ABB RAPID module: P800.mod

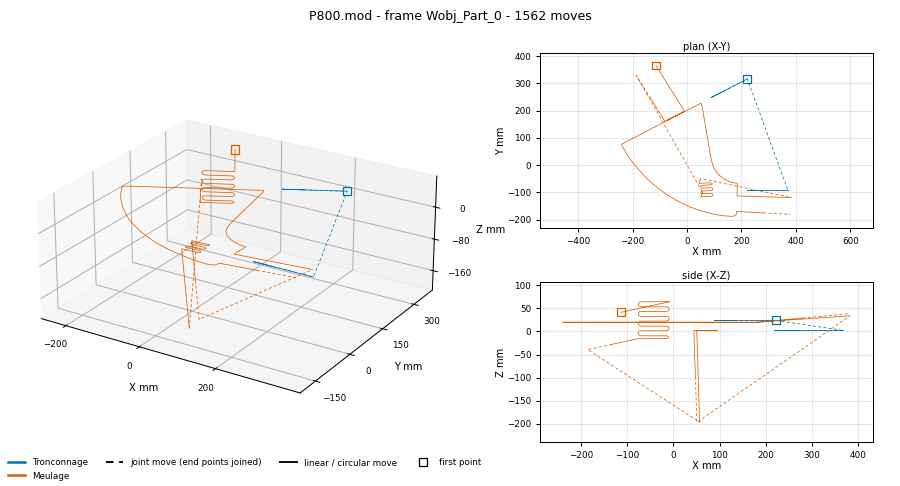
[picture p0: tool path of P800.mod in frame Wobj_Part_0, 1562 of 1576 moves have a stored position in this frame; points joined in program order, loops and branches not executed]
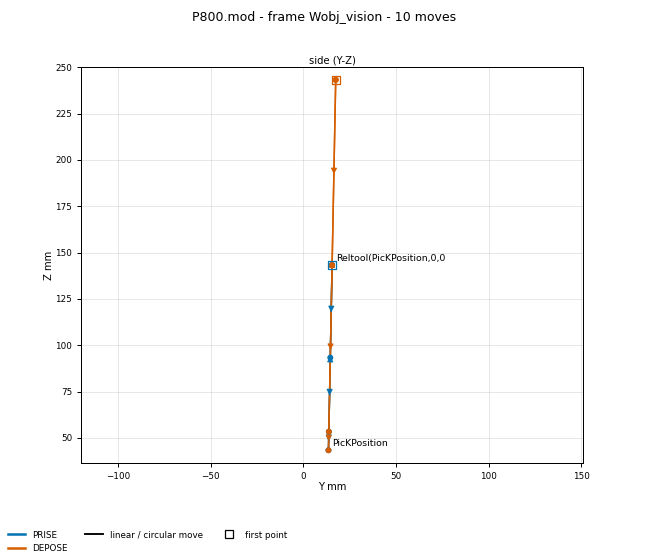
[picture p1: tool path of P800.mod in frame Wobj_vision, 10 of 1576 moves have a stored position in this frame; points joined in program order, loops and branches not executed]
MODULE P800

    ! Nom         :P800
    ! Description :
    ! Créé le     :31/05/2023 15:18:07

    LOCAL CONST SPEEDDATA VitesseLente :=[3,500,0,0];
	LOCAL CONST SPEEDDATA VitesseRapide :=[30,500,0,0];
	LOCAL CONST SPEEDDATA VitesseTronconnage :=[2,500,0,0];
	LOCAL CONST SPEEDDATA VitesseTronconnageApp :=[10,500,0,0];
    !
    !Point de prise
    LOCAL PERS Robtarget PicKPosition := [[-28.4505957143779,13.556706441967,43.2914417962046],[0.00189142649690449,0.425071382664564,-0.905103593114038,0.00991099780553871],[0,0,0,0],[8.999999E+09,8.999999E+09,8.999999E+09,8.999999E+09,8.999999E+09,8.999999E+09]];
	LOCAL PERS Pose Ref := [[0,0,0],[1,0,0,0]];
    !
    !Declaration des points de meulage

    !Tr_meulage_motif_1 : Meulage d'un motif
    LOCAL CONST Robtarget Tr_meulage_motif_1_0 := [[-8.6116181640625,197.027234375,64.58371875],[0.205457264684473,-0.183019148705642,0.639481640238406,-0.717881978735665],[0,0,0,0],[8.999999E+09,8.999999E+09,8.999999E+09,8.999999E+09,8.999999E+09,8.999999E+09]];
    LOCAL CONST Robtarget Tr_meulage_motif_1_1 := [[-9.49978125,196.567703125,64.58371875],[0.205457264684473,-0.183019148705642,0.639481640238406,-0.717881978735665],[0,0,0,0],[8.999999E+09,8.999999E+09,8.999999E+09,8.999999E+09,8.999999E+09,8.999999E+09]];
    LOCAL CONST Robtarget Tr_meulage_motif_1_2 := [[-10.3879453125,196.108171875,64.58371875],[0.205457264684473,-0.183019148705642,0.639481640238406,-0.717881978735665],[0,0,0,0],[8.999999E+09,8.999999E+09,8.999999E+09,8.999999E+09,8.999999E+09,8.999999E+09]];
    LOCAL CONST Robtarget Tr_meulage_motif_1_3 := [[-11.276109375,195.648640625,64.58371875],[0.205457264684473,-0.183019148705642,0.639481640238406,-0.717881978735665],[0,0,0,0],[8.999999E+09,8.999999E+09,8.999999E+09,8.999999E+09,8.999999E+09,8.999999E+09]];
    LOCAL CONST Robtarget Tr_meulage_motif_1_4 := [[-12.1642724609375,195.189125,64.58372265625],[0.205457264684473,-0.183019148705642,0.639481640238406,-0.717881978735665],[0,0,0,0],[8.999999E+09,8.999999E+09,8.999999E+09,8.999999E+09,8.999999E+09,8.999999E+09]];
    LOCAL CONST Robtarget Tr_meulage_motif_1_5 := [[-13.0524365234375,194.72959375,64.58372265625],[0.205457264684473,-0.183019148705642,0.639481640238406,-0.717881978735665],[0,0,0,0],[8.999999E+09,8.999999E+09,8.999999E+09,8.999999E+09,8.999999E+09,8.999999E+09]];
    LOCAL CONST Robtarget Tr_meulage_motif_1_6 := [[-13.940599609375,194.2700625,64.58372265625],[0.205457264684473,-0.183019148705642,0.639481640238406,-0.717881978735665],[0,0,0,0],[8.999999E+09,8.999999E+09,8.999999E+09,8.999999E+09,8.999999E+09,8.999999E+09]];
    LOCAL CONST Robtarget Tr_meulage_motif_1_7 := [[-14.828763671875,193.81053125,64.58372265625],[0.205457264684473,-0.183019148705642,0.639481640238406,-0.717881978735665],[0,0,0,0],[8.999999E+09,8.999999E+09,8.999999E+09,8.999999E+09,8.999999E+09,8.999999E+09]];
    LOCAL CONST Robtarget Tr_meulage_motif_1_8 := [[-15.7169267578125,193.351015625,64.58372265625],[0.205457264684473,-0.183019148705642,0.639481640238406,-0.717881978735665],[0,0,0,0],[8.999999E+09,8.999999E+09,8.999999E+09,8.999999E+09,8.999999E+09,8.999999E+09]];
    LOCAL CONST Robtarget Tr_meulage_motif_1_9 := [[-16.60508984375,192.891484375,64.58372265625],[0.205457264684473,-0.183019148705642,0.639481640238406,-0.717881978735665],[0,0,0,0],[8.999999E+09,8.999999E+09,8.999999E+09,8.999999E+09,8.999999E+09,8.999999E+09]];
    LOCAL CONST Robtarget Tr_meulage_motif_1_10 := [[-17.49325390625,192.431953125,64.58372265625],[0.205457264684473,-0.183019148705642,0.639481640238406,-0.717881978735665],[0,0,0,0],[8.999999E+09,8.999999E+09,8.999999E+09,8.999999E+09,8.999999E+09,8.999999E+09]];
    LOCAL CONST Robtarget Tr_meulage_motif_1_11 := [[-18.38141796875,191.972421875,64.58372265625],[0.205457264684473,-0.183019148705642,0.639481640238406,-0.717881978735665],[0,0,0,0],[8.999999E+09,8.999999E+09,8.999999E+09,8.999999E+09,8.999999E+09,8.999999E+09]];
    LOCAL CONST Robtarget Tr_meulage_motif_1_12 := [[-19.26958203125,191.51290625,64.5837265625],[0.205457264684473,-0.183019148705642,0.639481640238406,-0.717881978735665],[0,0,0,0],[8.999999E+09,8.999999E+09,8.999999E+09,8.999999E+09,8.999999E+09,8.999999E+09]];
    LOCAL CONST Robtarget Tr_meulage_motif_1_13 := [[-20.157744140625,191.053375,64.5837265625],[0.205457264684473,-0.183019148705642,0.639481640238406,-0.717881978735665],[0,0,0,0],[8.999999E+09,8.999999E+09,8.999999E+09,8.999999E+09,8.999999E+09,8.999999E+09]];
    LOCAL CONST Robtarget Tr_meulage_motif_1_14 := [[-21.045908203125,190.59384375,64.5837265625],[0.205457264684473,-0.183019148705642,0.639481640238406,-0.717881978735665],[0,0,0,0],[8.999999E+09,8.999999E+09,8.999999E+09,8.999999E+09,8.999999E+09,8.999999E+09]];
    LOCAL CONST Robtarget Tr_meulage_motif_1_15 := [[-21.934072265625,190.1343125,64.5837265625],[0.205457264684473,-0.183019148705642,0.639481640238406,-0.717881978735665],[0,0,0,0],[8.999999E+09,8.999999E+09,8.999999E+09,8.999999E+09,8.999999E+09,8.999999E+09]];
    LOCAL CONST Robtarget Tr_meulage_motif_1_16 := [[-22.822236328125,189.674796875,64.5837265625],[0.205457264684473,-0.183019148705642,0.639481640238406,-0.717881978735665],[0,0,0,0],[8.999999E+09,8.999999E+09,8.999999E+09,8.999999E+09,8.999999E+09,8.999999E+09]];
    LOCAL CONST Robtarget Tr_meulage_motif_1_17 := [[-23.7103984375,189.215265625,64.5837265625],[0.205457264684473,-0.183019148705642,0.639481640238406,-0.717881978735665],[0,0,0,0],[8.999999E+09,8.999999E+09,8.999999E+09,8.999999E+09,8.999999E+09,8.999999E+09]];
    LOCAL CONST Robtarget Tr_meulage_motif_1_18 := [[-24.5985625,188.755734375,64.5837265625],[0.205457264684473,-0.183019148705642,0.639481640238406,-0.717881978735665],[0,0,0,0],[8.999999E+09,8.999999E+09,8.999999E+09,8.999999E+09,8.999999E+09,8.999999E+09]];
    LOCAL CONST Robtarget Tr_meulage_motif_1_19 := [[-25.4867265625,188.296203125,64.5837265625],[0.205457264684473,-0.183019148705642,0.639481640238406,-0.717881978735665],[0,0,0,0],[8.999999E+09,8.999999E+09,8.999999E+09,8.999999E+09,8.999999E+09,8.999999E+09]];
    LOCAL CONST Robtarget Tr_meulage_motif_1_20 := [[-26.374890625,187.8366875,64.5837265625],[0.205457264684473,-0.183019148705642,0.639481640238406,-0.717881978735665],[0,0,0,0],[8.999999E+09,8.999999E+09,8.999999E+09,8.999999E+09,8.999999E+09,8.999999E+09]];
    LOCAL CONST Robtarget Tr_meulage_motif_1_21 := [[-27.263052734375,187.37715625,64.58373046875],[0.205457264684473,-0.183019148705642,0.639481640238406,-0.717881978735665],[0,0,0,0],[8.999999E+09,8.999999E+09,8.999999E+09,8.999999E+09,8.999999E+09,8.999999E+09]];
    LOCAL CONST Robtarget Tr_meulage_motif_1_22 := [[-28.151216796875,186.917625,64.58373046875],[0.205457264684473,-0.183019148705642,0.639481640238406,-0.717881978735665],[0,0,0,0],[8.999999E+09,8.999999E+09,8.999999E+09,8.999999E+09,8.999999E+09,8.999999E+09]];
    LOCAL CONST Robtarget Tr_meulage_motif_1_23 := [[-29.039380859375,186.45809375,64.58373046875],[0.205457264684473,-0.183019148705642,0.639481640238406,-0.717881978735665],[0,0,0,0],[8.999999E+09,8.999999E+09,8.999999E+09,8.999999E+09,8.999999E+09,8.999999E+09]];
    LOCAL CONST Robtarget Tr_meulage_motif_1_24 := [[-29.927544921875,185.9985625,64.58373046875],[0.205457264684473,-0.183019148705642,0.639481640238406,-0.717881978735665],[0,0,0,0],[8.999999E+09,8.999999E+09,8.999999E+09,8.999999E+09,8.999999E+09,8.999999E+09]];
    LOCAL CONST Robtarget Tr_meulage_motif_1_25 := [[-30.815708984375,185.539046875,64.58373046875],[0.205457264684473,-0.183019148705642,0.639481640238406,-0.717881978735665],[0,0,0,0],[8.999999E+09,8.999999E+09,8.999999E+09,8.999999E+09,8.999999E+09,8.999999E+09]];
    LOCAL CONST Robtarget Tr_meulage_motif_1_26 := [[-31.70387109375,185.079515625,64.58373046875],[0.205457264684473,-0.183019148705642,0.639481640238406,-0.717881978735665],[0,0,0,0],[8.999999E+09,8.999999E+09,8.999999E+09,8.999999E+09,8.999999E+09,8.999999E+09]];
    LOCAL CONST Robtarget Tr_meulage_motif_1_27 := [[-32.59203515625,184.619984375,64.58373046875],[0.205457264684473,-0.183019148705642,0.639481640238406,-0.717881978735665],[0,0,0,0],[8.999999E+09,8.999999E+09,8.999999E+09,8.999999E+09,8.999999E+09,8.999999E+09]];
    LOCAL CONST Robtarget Tr_meulage_motif_1_28 := [[-33.48019921875,184.160453125,64.58373046875],[0.205457264684473,-0.183019148705642,0.639481640238406,-0.717881978735665],[0,0,0,0],[8.999999E+09,8.999999E+09,8.999999E+09,8.999999E+09,8.999999E+09,8.999999E+09]];
    LOCAL CONST Robtarget Tr_meulage_motif_1_29 := [[-34.36836328125,183.7009375,64.583734375],[0.205457264684473,-0.183019148705642,0.639481640238406,-0.717881978735665],[0,0,0,0],[8.999999E+09,8.999999E+09,8.999999E+09,8.999999E+09,8.999999E+09,8.999999E+09]];
    LOCAL CONST Robtarget Tr_meulage_motif_1_30 := [[-35.25652734375,183.24140625,64.583734375],[0.205457264684473,-0.183019148705642,0.639481640238406,-0.717881978735665],[0,0,0,0],[8.999999E+09,8.999999E+09,8.999999E+09,8.999999E+09,8.999999E+09,8.999999E+09]];
    LOCAL CONST Robtarget Tr_meulage_motif_1_31 := [[-36.14469140625,182.781875,64.583734375],[0.205457264684473,-0.183019148705642,0.639481640238406,-0.717881978735665],[0,0,0,0],[8.999999E+09,8.999999E+09,8.999999E+09,8.999999E+09,8.999999E+09,8.999999E+09]];
    LOCAL CONST Robtarget Tr_meulage_motif_1_32 := [[-37.0328515625,182.32234375,64.583734375],[0.205457264684473,-0.183019148705642,0.639481640238406,-0.717881978735665],[0,0,0,0],[8.999999E+09,8.999999E+09,8.999999E+09,8.999999E+09,8.999999E+09,8.999999E+09]];
    LOCAL CONST Robtarget Tr_meulage_motif_1_33 := [[-37.921015625,181.862828125,64.583734375],[0.205457264684473,-0.183019148705642,0.639481640238406,-0.717881978735665],[0,0,0,0],[8.999999E+09,8.999999E+09,8.999999E+09,8.999999E+09,8.999999E+09,8.999999E+09]];
    LOCAL CONST Robtarget Tr_meulage_motif_1_34 := [[-38.8091796875,181.403296875,64.583734375],[0.205457264684473,-0.183019148705642,0.639481640238406,-0.717881978735665],[0,0,0,0],[8.999999E+09,8.999999E+09,8.999999E+09,8.999999E+09,8.999999E+09,8.999999E+09]];
    LOCAL CONST Robtarget Tr_meulage_motif_1_35 := [[-39.69734375,180.943765625,64.583734375],[0.205457264684473,-0.183019148705642,0.639481640238406,-0.717881978735665],[0,0,0,0],[8.999999E+09,8.999999E+09,8.999999E+09,8.999999E+09,8.999999E+09,8.999999E+09]];
    LOCAL CONST Robtarget Tr_meulage_motif_1_36 := [[-40.5855078125,180.484234375,64.583734375],[0.205457264684473,-0.183019148705642,0.639481640238406,-0.717881978735665],[0,0,0,0],[8.999999E+09,8.999999E+09,8.999999E+09,8.999999E+09,8.999999E+09,8.999999E+09]];
    LOCAL CONST Robtarget Tr_meulage_motif_1_37 := [[-41.473671875,180.02471875,64.583734375],[0.205457264684473,-0.183019148705642,0.639481640238406,-0.717881978735665],[0,0,0,0],[8.999999E+09,8.999999E+09,8.999999E+09,8.999999E+09,8.999999E+09,8.999999E+09]];
    LOCAL CONST Robtarget Tr_meulage_motif_1_38 := [[-42.3618359375,179.5651875,64.58373828125],[0.205457264684473,-0.183019148705642,0.639481640238406,-0.717881978735665],[0,0,0,0],[8.999999E+09,8.999999E+09,8.999999E+09,8.999999E+09,8.999999E+09,8.999999E+09]];
    LOCAL CONST Robtarget Tr_meulage_motif_1_39 := [[-43.25,179.10565625,64.58373828125],[0.205457264684473,-0.183019148705642,0.639481640238406,-0.717881978735665],[0,0,0,0],[8.999999E+09,8.999999E+09,8.999999E+09,8.999999E+09,8.999999E+09,8.999999E+09]];
    LOCAL CONST Robtarget Tr_meulage_motif_1_40 := [[-44.13816015625,178.646125,64.58373828125],[0.205457264684473,-0.183019148705642,0.639481640238406,-0.717881978735665],[0,0,0,0],[8.999999E+09,8.999999E+09,8.999999E+09,8.999999E+09,8.999999E+09,8.999999E+09]];
    LOCAL CONST Robtarget Tr_meulage_motif_1_41 := [[-45.02632421875,178.186609375,64.58373828125],[0.205457264684473,-0.183019148705642,0.639481640238406,-0.717881978735665],[0,0,0,0],[8.999999E+09,8.999999E+09,8.999999E+09,8.999999E+09,8.999999E+09,8.999999E+09]];
    LOCAL CONST Robtarget Tr_meulage_motif_1_42 := [[-45.91448828125,177.727078125,64.58373828125],[0.205457264684473,-0.183019148705642,0.639481640238406,-0.717881978735665],[0,0,0,0],[8.999999E+09,8.999999E+09,8.999999E+09,8.999999E+09,8.999999E+09,8.999999E+09]];
    LOCAL CONST Robtarget Tr_meulage_motif_1_43 := [[-46.80265234375,177.267546875,64.58373828125],[0.205457264684473,-0.183019148705642,0.639481640238406,-0.717881978735665],[0,0,0,0],[8.999999E+09,8.999999E+09,8.999999E+09,8.999999E+09,8.999999E+09,8.999999E+09]];
    LOCAL CONST Robtarget Tr_meulage_motif_1_44 := [[-47.69081640625,176.808015625,64.58373828125],[0.205457264684473,-0.183019148705642,0.639481640238406,-0.717881978735665],[0,0,0,0],[8.999999E+09,8.999999E+09,8.999999E+09,8.999999E+09,8.999999E+09,8.999999E+09]];
    LOCAL CONST Robtarget Tr_meulage_motif_1_45 := [[-48.57898046875,176.3485,64.58373828125],[0.205457264684473,-0.183019148705642,0.639481640238406,-0.717881978735665],[0,0,0,0],[8.999999E+09,8.999999E+09,8.999999E+09,8.999999E+09,8.999999E+09,8.999999E+09]];
    LOCAL CONST Robtarget Tr_meulage_motif_1_46 := [[-49.46714453125,175.88896875,64.5837421875],[0.205457264684473,-0.183019148705642,0.639481640238406,-0.717881978735665],[0,0,0,0],[8.999999E+09,8.999999E+09,8.999999E+09,8.999999E+09,8.999999E+09,8.999999E+09]];
    LOCAL CONST Robtarget Tr_meulage_motif_1_47 := [[-50.35530859375,175.4294375,64.5837421875],[0.205457264684473,-0.183019148705642,0.639481640238406,-0.717881978735665],[0,0,0,0],[8.999999E+09,8.999999E+09,8.999999E+09,8.999999E+09,8.999999E+09,8.999999E+09]];
    LOCAL CONST Robtarget Tr_meulage_motif_1_48 := [[-51.24347265625,174.96990625,64.5837421875],[0.205457264684473,-0.183019148705642,0.639481640238406,-0.717881978735665],[0,0,0,0],[8.999999E+09,8.999999E+09,8.999999E+09,8.999999E+09,8.999999E+09,8.999999E+09]];
    LOCAL CONST Robtarget Tr_meulage_motif_1_49 := [[-52.1316328125,174.510390625,64.5837421875],[0.205457264684473,-0.183019148705642,0.639481640238406,-0.717881978735665],[0,0,0,0],[8.999999E+09,8.999999E+09,8.999999E+09,8.999999E+09,8.999999E+09,8.999999E+09]];
    LOCAL CONST Robtarget Tr_meulage_motif_1_50 := [[-53.019796875,174.050859375,64.5837421875],[0.205457264684473,-0.183019148705642,0.639481640238406,-0.717881978735665],[0,0,0,0],[8.999999E+09,8.999999E+09,8.999999E+09,8.999999E+09,8.999999E+09,8.999999E+09]];
    LOCAL CONST Robtarget Tr_meulage_motif_1_51 := [[-53.9079609375,173.591328125,64.5837421875],[0.205457264684473,-0.183019148705642,0.639481640238406,-0.717881978735665],[0,0,0,0],[8.999999E+09,8.999999E+09,8.999999E+09,8.999999E+09,8.999999E+09,8.999999E+09]];
    LOCAL CONST Robtarget Tr_meulage_motif_1_52 := [[-54.796125,173.131796875,64.5837421875],[0.205457264684473,-0.183019148705642,0.639481640238406,-0.717881978735665],[0,0,0,0],[8.999999E+09,8.999999E+09,8.999999E+09,8.999999E+09,8.999999E+09,8.999999E+09]];
    LOCAL CONST Robtarget Tr_meulage_motif_1_53 := [[-55.6842890625,172.67228125,64.5837421875],[0.205457264684473,-0.183019148705642,0.639481640238406,-0.717881978735665],[0,0,0,0],[8.999999E+09,8.999999E+09,8.999999E+09,8.999999E+09,8.999999E+09,8.999999E+09]];
    LOCAL CONST Robtarget Tr_meulage_motif_1_54 := [[-56.572453125,172.21275,64.5837421875],[0.205457264684473,-0.183019148705642,0.639481640238406,-0.717881978735665],[0,0,0,0],[8.999999E+09,8.999999E+09,8.999999E+09,8.999999E+09,8.999999E+09,8.999999E+09]];
    LOCAL CONST Robtarget Tr_meulage_motif_1_55 := [[-57.4606171875,171.75321875,64.58374609375],[0.205457264684473,-0.183019148705642,0.639481640238406,-0.717881978735665],[0,0,0,0],[8.999999E+09,8.999999E+09,8.999999E+09,8.999999E+09,8.999999E+09,8.999999E+09]];
    LOCAL CONST Robtarget Tr_meulage_motif_1_56 := [[-58.34878125,171.2936875,64.58374609375],[0.205457264684473,-0.183019148705642,0.639481640238406,-0.717881978735665],[0,0,0,0],[8.999999E+09,8.999999E+09,8.999999E+09,8.999999E+09,8.999999E+09,8.999999E+09]];
    LOCAL CONST Robtarget Tr_meulage_motif_1_57 := [[-59.23694140625,170.834171875,64.58374609375],[0.205457264684473,-0.183019148705642,0.639481640238406,-0.717881978735665],[0,0,0,0],[8.999999E+09,8.999999E+09,8.999999E+09,8.999999E+09,8.999999E+09,8.999999E+09]];
    LOCAL CONST Robtarget Tr_meulage_motif_1_58 := [[-60.12510546875,170.374640625,64.58374609375],[0.205457264684473,-0.183019148705642,0.639481640238406,-0.717881978735665],[0,0,0,0],[8.999999E+09,8.999999E+09,8.999999E+09,8.999999E+09,8.999999E+09,8.999999E+09]];
    LOCAL CONST Robtarget Tr_meulage_motif_1_59 := [[-61.01326953125,169.915109375,64.58374609375],[0.205457264684473,-0.183019148705642,0.639481640238406,-0.717881978735665],[0,0,0,0],[8.999999E+09,8.999999E+09,8.999999E+09,8.999999E+09,8.999999E+09,8.999999E+09]];
    LOCAL CONST Robtarget Tr_meulage_motif_1_60 := [[-61.90143359375,169.455578125,64.58374609375],[0.205457264684473,-0.183019148705642,0.639481640238406,-0.717881978735665],[0,0,0,0],[8.999999E+09,8.999999E+09,8.999999E+09,8.999999E+09,8.999999E+09,8.999999E+09]];
    LOCAL CONST Robtarget Tr_meulage_motif_1_61 := [[-62.78959765625,168.9960625,64.58374609375],[0.205457264684473,-0.183019148705642,0.639481640238406,-0.717881978735665],[0,0,0,0],[8.999999E+09,8.999999E+09,8.999999E+09,8.999999E+09,8.999999E+09,8.999999E+09]];
    LOCAL CONST Robtarget Tr_meulage_motif_1_62 := [[-63.67776171875,168.53653125,64.58374609375],[0.205457264684473,-0.183019148705642,0.639481640238406,-0.717881978735665],[0,0,0,0],[8.999999E+09,8.999999E+09,8.999999E+09,8.999999E+09,8.999999E+09,8.999999E+09]];
    LOCAL CONST Robtarget Tr_meulage_motif_1_63 := [[-64.56592578125,168.077,64.58374609375],[0.205457264684473,-0.183019148705642,0.639481640238406,-0.717881978735665],[0,0,0,0],[8.999999E+09,8.999999E+09,8.999999E+09,8.999999E+09,8.999999E+09,8.999999E+09]];
    LOCAL CONST Robtarget Tr_meulage_motif_1_64 := [[-65.45408984375,167.61746875,64.58375],[0.205457264684473,-0.183019148705642,0.639481640238406,-0.717881978735665],[0,0,0,0],[8.999999E+09,8.999999E+09,8.999999E+09,8.999999E+09,8.999999E+09,8.999999E+09]];
    LOCAL CONST Robtarget Tr_meulage_motif_1_65 := [[-66.34225,167.157953125,64.58375],[0.205457264684473,-0.183019148705642,0.639481640238406,-0.717881978735665],[0,0,0,0],[8.999999E+09,8.999999E+09,8.999999E+09,8.999999E+09,8.999999E+09,8.999999E+09]];
    LOCAL CONST Robtarget Tr_meulage_motif_1_66 := [[-67.2304140625,166.698421875,64.58375],[0.205457264684473,-0.183019148705642,0.639481640238406,-0.717881978735665],[0,0,0,0],[8.999999E+09,8.999999E+09,8.999999E+09,8.999999E+09,8.999999E+09,8.999999E+09]];
    LOCAL CONST Robtarget Tr_meulage_motif_1_67 := [[-68.118578125,166.238890625,64.58375],[0.205457264684473,-0.183019148705642,0.639481640238406,-0.717881978735665],[0,0,0,0],[8.999999E+09,8.999999E+09,8.999999E+09,8.999999E+09,8.999999E+09,8.999999E+09]];
    LOCAL CONST Robtarget Tr_meulage_motif_1_68 := [[-69.0067421875,165.779359375,64.58375],[0.205457264684473,-0.183019148705642,0.639481640238406,-0.717881978735665],[0,0,0,0],[8.999999E+09,8.999999E+09,8.999999E+09,8.999999E+09,8.999999E+09,8.999999E+09]];
    LOCAL CONST Robtarget Tr_meulage_motif_1_69 := [[-69.89490625,165.31984375,64.58375],[0.205457264684473,-0.183019148705642,0.639481640238406,-0.717881978735665],[0,0,0,0],[8.999999E+09,8.999999E+09,8.999999E+09,8.999999E+09,8.999999E+09,8.999999E+09]];
    LOCAL CONST Robtarget Tr_meulage_motif_1_70 := [[-70.7768671875,164.864515625,64.47316015625],[0.205457264684473,-0.183019148705642,0.639481640238406,-0.717881978735665],[0,0,0,0],[8.999999E+09,8.999999E+09,8.999999E+09,8.999999E+09,8.999999E+09,8.999999E+09]];
    LOCAL CONST Robtarget Tr_meulage_motif_1_71 := [[-71.6182890625,164.4310625,64.26198046875],[0.205457264684473,-0.183019148705642,0.639481640238406,-0.717881978735665],[0,0,0,0],[8.999999E+09,8.999999E+09,8.999999E+09,8.999999E+09,8.999999E+09,8.999999E+09]];
    LOCAL CONST Robtarget Tr_meulage_motif_1_72 := [[-72.376640625,164.041140625,63.99014453125],[0.205457264684473,-0.183019148705642,0.639481640238406,-0.717881978735665],[0,0,0,0],[8.999999E+09,8.999999E+09,8.999999E+09,8.999999E+09,8.999999E+09,8.999999E+09]];
    LOCAL CONST Robtarget Tr_meulage_motif_1_73 := [[-73.0436875,163.698484375,63.71421875],[0.205457264684473,-0.183019148705642,0.639481640238406,-0.717881978735665],[0,0,0,0],[8.999999E+09,8.999999E+09,8.999999E+09,8.999999E+09,8.999999E+09,8.999999E+09]];
    LOCAL CONST Robtarget Tr_meulage_motif_1_74 := [[-74.0238984375,163.196859375,63.09811328125],[0.205457264684473,-0.183019148705642,0.639481640238406,-0.717881978735665],[0,0,0,0],[8.999999E+09,8.999999E+09,8.999999E+09,8.999999E+09,8.999999E+09,8.999999E+09]];
    LOCAL CONST Robtarget Tr_meulage_motif_1_75 := [[-74.9363671875,162.732359375,62.250484375],[0.205457264684473,-0.183019148705642,0.639481640238406,-0.717881978735665],[0,0,0,0],[8.999999E+09,8.999999E+09,8.999999E+09,8.999999E+09,8.999999E+09,8.999999E+09]];
    LOCAL CONST Robtarget Tr_meulage_motif_1_76 := [[-75.6929765625,162.35009375,61.226640625],[0.205457264684473,-0.183019148705642,0.639481640238406,-0.717881978735665],[0,0,0,0],[8.999999E+09,8.999999E+09,8.999999E+09,8.999999E+09,8.999999E+09,8.999999E+09]];
    LOCAL CONST Robtarget Tr_meulage_motif_1_77 := [[-76.130625,162.133671875,60.11048828125],[0.205457264684473,-0.183019148705642,0.639481640238406,-0.717881978735665],[0,0,0,0],[8.999999E+09,8.999999E+09,8.999999E+09,8.999999E+09,8.999999E+09,8.999999E+09]];
    LOCAL CONST Robtarget Tr_meulage_motif_1_78 := [[-76.1572109375,162.12615625,59.41454296875],[0.205457264684473,-0.183019148705642,0.639481640238406,-0.717881978735665],[0,0,0,0],[8.999999E+09,8.999999E+09,8.999999E+09,8.999999E+09,8.999999E+09,8.999999E+09]];
    LOCAL CONST Robtarget Tr_meulage_motif_1_79 := [[-76.1596328125,162.130828125,58.7533125],[0.205457264684473,-0.183019148705642,0.639481640238406,-0.717881978735665],[0,0,0,0],[8.999999E+09,8.999999E+09,8.999999E+09,8.999999E+09,8.999999E+09,8.999999E+09]];
    LOCAL CONST Robtarget Tr_meulage_motif_1_80 := [[-76.1133125,162.160734375,58.0922421875],[0.205457264684473,-0.183019148705642,0.639481640238406,-0.717881978735665],[0,0,0,0],[8.999999E+09,8.999999E+09,8.999999E+09,8.999999E+09,8.999999E+09,8.999999E+09]];
    LOCAL CONST Robtarget Tr_meulage_motif_1_81 := [[-75.67484375,162.39746875,56.99052734375],[0.205457264684473,-0.183019148705642,0.639481640238406,-0.717881978735665],[0,0,0,0],[8.999999E+09,8.999999E+09,8.999999E+09,8.999999E+09,8.999999E+09,8.999999E+09]];
    LOCAL CONST Robtarget Tr_meulage_motif_1_82 := [[-74.9177109375,162.798234375,55.98393359375],[0.205457264684473,-0.183019148705642,0.639481640238406,-0.717881978735665],[0,0,0,0],[8.999999E+09,8.999999E+09,8.999999E+09,8.999999E+09,8.999999E+09,8.999999E+09]];
    LOCAL CONST Robtarget Tr_meulage_motif_1_83 := [[-74.011765625,163.274390625,55.15508203125],[0.205457264684473,-0.183019148705642,0.639481640238406,-0.717881978735665],[0,0,0,0],[8.999999E+09,8.999999E+09,8.999999E+09,8.999999E+09,8.999999E+09,8.999999E+09]];
    LOCAL CONST Robtarget Tr_meulage_motif_1_84 := [[-73.4029921875,163.592921875,54.75934375],[0.205457264684473,-0.183019148705642,0.639481640238406,-0.717881978735665],[0,0,0,0],[8.999999E+09,8.999999E+09,8.999999E+09,8.999999E+09,8.999999E+09,8.999999E+09]];
    LOCAL CONST Robtarget Tr_meulage_motif_1_85 := [[-72.376140625,164.128578125,54.271828125],[0.205457264684473,-0.183019148705642,0.639481640238406,-0.717881978735665],[0,0,0,0],[8.999999E+09,8.999999E+09,8.999999E+09,8.999999E+09,8.999999E+09,8.999999E+09]];
    LOCAL CONST Robtarget Tr_meulage_motif_1_86 := [[-71.6265859375,164.518765625,54.0077421875],[0.205457264684473,-0.183019148705642,0.639481640238406,-0.717881978735665],[0,0,0,0],[8.999999E+09,8.999999E+09,8.999999E+09,8.999999E+09,8.999999E+09,8.999999E+09]];
    LOCAL CONST Robtarget Tr_meulage_motif_1_87 := [[-70.7995625,164.948484375,53.80328125],[0.205457264684473,-0.183019148705642,0.639481640238406,-0.717881978735665],[0,0,0,0],[8.999999E+09,8.999999E+09,8.999999E+09,8.999999E+09,8.999999E+09,8.999999E+09]];
    LOCAL CONST Robtarget Tr_meulage_motif_1_88 := [[-69.928171875,165.4003125,53.69469140625],[0.205457264684473,-0.183019148705642,0.639481640238406,-0.717881978735665],[0,0,0,0],[8.999999E+09,8.999999E+09,8.999999E+09,8.999999E+09,8.999999E+09,8.999999E+09]];
    LOCAL CONST Robtarget Tr_meulage_motif_1_89 := [[-69.0470234375,165.857203125,53.58409765625],[0.205457264684473,-0.183019148705642,0.639481640238406,-0.717881978735665],[0,0,0,0],[8.999999E+09,8.999999E+09,8.999999E+09,8.999999E+09,8.999999E+09,8.999999E+09]];
    LOCAL CONST Robtarget Tr_meulage_motif_1_90 := [[-68.158859375,166.316734375,53.58409765625],[0.205457264684473,-0.183019148705642,0.639481640238406,-0.717881978735665],[0,0,0,0],[8.999999E+09,8.999999E+09,8.999999E+09,8.999999E+09,8.999999E+09,8.999999E+09]];
    LOCAL CONST Robtarget Tr_meulage_motif_1_91 := [[-67.2706953125,166.77625,53.58409765625],[0.205457264684473,-0.183019148705642,0.639481640238406,-0.717881978735665],[0,0,0,0],[8.999999E+09,8.999999E+09,8.999999E+09,8.999999E+09,8.999999E+09,8.999999E+09]];
    LOCAL CONST Robtarget Tr_meulage_motif_1_92 := [[-66.38253125,167.23578125,53.58409765625],[0.205457264684473,-0.183019148705642,0.639481640238406,-0.717881978735665],[0,0,0,0],[8.999999E+09,8.999999E+09,8.999999E+09,8.999999E+09,8.999999E+09,8.999999E+09]];
    LOCAL CONST Robtarget Tr_meulage_motif_1_93 := [[-65.4943671875,167.6953125,53.58409765625],[0.205457264684473,-0.183019148705642,0.639481640238406,-0.717881978735665],[0,0,0,0],[8.999999E+09,8.999999E+09,8.999999E+09,8.999999E+09,8.999999E+09,8.999999E+09]];
    LOCAL CONST Robtarget Tr_meulage_motif_1_94 := [[-64.606203125,168.15484375,53.58409765625],[0.205457264684473,-0.183019148705642,0.639481640238406,-0.717881978735665],[0,0,0,0],[8.999999E+09,8.999999E+09,8.999999E+09,8.999999E+09,8.999999E+09,8.999999E+09]];
    LOCAL CONST Robtarget Tr_meulage_motif_1_95 := [[-63.7180390625,168.614359375,53.58409765625],[0.205457264684473,-0.183019148705642,0.639481640238406,-0.717881978735665],[0,0,0,0],[8.999999E+09,8.999999E+09,8.999999E+09,8.999999E+09,8.999999E+09,8.999999E+09]];
    LOCAL CONST Robtarget Tr_meulage_motif_1_96 := [[-62.829875,169.073890625,53.58409765625],[0.205457264684473,-0.183019148705642,0.639481640238406,-0.717881978735665],[0,0,0,0],[8.999999E+09,8.999999E+09,8.999999E+09,8.999999E+09,8.999999E+09,8.999999E+09]];
    LOCAL CONST Robtarget Tr_meulage_motif_1_97 := [[-61.9417109375,169.533421875,53.58409765625],[0.205457264684473,-0.183019148705642,0.639481640238406,-0.717881978735665],[0,0,0,0],[8.999999E+09,8.999999E+09,8.999999E+09,8.999999E+09,8.999999E+09,8.999999E+09]];
    LOCAL CONST Robtarget Tr_meulage_motif_1_98 := [[-61.053546875,169.992953125,53.58409375],[0.205457264684473,-0.183019148705642,0.639481640238406,-0.717881978735665],[0,0,0,0],[8.999999E+09,8.999999E+09,8.999999E+09,8.999999E+09,8.999999E+09,8.999999E+09]];
    LOCAL CONST Robtarget Tr_meulage_motif_1_99 := [[-60.1653828125,170.45246875,53.58409375],[0.205457264684473,-0.183019148705642,0.639481640238406,-0.717881978735665],[0,0,0,0],[8.999999E+09,8.999999E+09,8.999999E+09,8.999999E+09,8.999999E+09,8.999999E+09]];
    LOCAL CONST Robtarget Tr_meulage_motif_1_100 := [[-59.27721875,170.912,53.58409375],[0.205457264684473,-0.183019148705642,0.639481640238406,-0.717881978735665],[0,0,0,0],[8.999999E+09,8.999999E+09,8.999999E+09,8.999999E+09,8.999999E+09,8.999999E+09]];
    LOCAL CONST Robtarget Tr_meulage_motif_1_101 := [[-58.38905859375,171.37153125,53.58409375],[0.205457264684473,-0.183019148705642,0.639481640238406,-0.717881978735665],[0,0,0,0],[8.999999E+09,8.999999E+09,8.999999E+09,8.999999E+09,8.999999E+09,8.999999E+09]];
    LOCAL CONST Robtarget Tr_meulage_motif_1_102 := [[-57.50089453125,171.8310625,53.58409375],[0.205457264684473,-0.183019148705642,0.639481640238406,-0.717881978735665],[0,0,0,0],[8.999999E+09,8.999999E+09,8.999999E+09,8.999999E+09,8.999999E+09,8.999999E+09]];
    LOCAL CONST Robtarget Tr_meulage_motif_1_103 := [[-56.61273046875,172.290578125,53.58409375],[0.205457264684473,-0.183019148705642,0.639481640238406,-0.717881978735665],[0,0,0,0],[8.999999E+09,8.999999E+09,8.999999E+09,8.999999E+09,8.999999E+09,8.999999E+09]];
    LOCAL CONST Robtarget Tr_meulage_motif_1_104 := [[-55.72456640625,172.750109375,53.58409375],[0.205457264684473,-0.183019148705642,0.639481640238406,-0.717881978735665],[0,0,0,0],[8.999999E+09,8.999999E+09,8.999999E+09,8.999999E+09,8.999999E+09,8.999999E+09]];
    LOCAL CONST Robtarget Tr_meulage_motif_1_105 := [[-54.83640234375,173.209640625,53.58409375],[0.205457264684473,-0.183019148705642,0.639481640238406,-0.717881978735665],[0,0,0,0],[8.999999E+09,8.999999E+09,8.999999E+09,8.999999E+09,8.999999E+09,8.999999E+09]];
    LOCAL CONST Robtarget Tr_meulage_motif_1_106 := [[-53.94823828125,173.669171875,53.58408984375],[0.205457264684473,-0.183019148705642,0.639481640238406,-0.717881978735665],[0,0,0,0],[8.999999E+09,8.999999E+09,8.999999E+09,8.999999E+09,8.999999E+09,8.999999E+09]];
    LOCAL CONST Robtarget Tr_meulage_motif_1_107 := [[-53.06007421875,174.1286875,53.58408984375],[0.205457264684473,-0.183019148705642,0.639481640238406,-0.717881978735665],[0,0,0,0],[8.999999E+09,8.999999E+09,8.999999E+09,8.999999E+09,8.999999E+09,8.999999E+09]];
    LOCAL CONST Robtarget Tr_meulage_motif_1_108 := [[-52.17191015625,174.58821875,53.58408984375],[0.205457264684473,-0.183019148705642,0.639481640238406,-0.717881978735665],[0,0,0,0],[8.999999E+09,8.999999E+09,8.999999E+09,8.999999E+09,8.999999E+09,8.999999E+09]];
    LOCAL CONST Robtarget Tr_meulage_motif_1_109 := [[-51.28375,175.04775,53.58408984375],[0.205457264684473,-0.183019148705642,0.639481640238406,-0.717881978735665],[0,0,0,0],[8.999999E+09,8.999999E+09,8.999999E+09,8.999999E+09,8.999999E+09,8.999999E+09]];
    LOCAL CONST Robtarget Tr_meulage_motif_1_110 := [[-50.3955859375,175.50728125,53.58408984375],[0.205457264684473,-0.183019148705642,0.639481640238406,-0.717881978735665],[0,0,0,0],[8.999999E+09,8.999999E+09,8.999999E+09,8.999999E+09,8.999999E+09,8.999999E+09]];
    LOCAL CONST Robtarget Tr_meulage_motif_1_111 := [[-49.507421875,175.966796875,53.58408984375],[0.205457264684473,-0.183019148705642,0.639481640238406,-0.717881978735665],[0,0,0,0],[8.999999E+09,8.999999E+09,8.999999E+09,8.999999E+09,8.999999E+09,8.999999E+09]];
    LOCAL CONST Robtarget Tr_meulage_motif_1_112 := [[-48.6192578125,176.426328125,53.58408984375],[0.205457264684473,-0.183019148705642,0.639481640238406,-0.717881978735665],[0,0,0,0],[8.999999E+09,8.999999E+09,8.999999E+09,8.999999E+09,8.999999E+09,8.999999E+09]];
    LOCAL CONST Robtarget Tr_meulage_motif_1_113 := [[-47.73109375,176.885859375,53.58408984375],[0.205457264684473,-0.183019148705642,0.639481640238406,-0.717881978735665],[0,0,0,0],[8.999999E+09,8.999999E+09,8.999999E+09,8.999999E+09,8.999999E+09,8.999999E+09]];
    LOCAL CONST Robtarget Tr_meulage_motif_1_114 := [[-46.8429296875,177.345390625,53.58408984375],[0.205457264684473,-0.183019148705642,0.639481640238406,-0.717881978735665],[0,0,0,0],[8.999999E+09,8.999999E+09,8.999999E+09,8.999999E+09,8.999999E+09,8.999999E+09]];
    LOCAL CONST Robtarget Tr_meulage_motif_1_115 := [[-45.954765625,177.80490625,53.5840859375],[0.205457264684473,-0.183019148705642,0.639481640238406,-0.717881978735665],[0,0,0,0],[8.999999E+09,8.999999E+09,8.999999E+09,8.999999E+09,8.999999E+09,8.999999E+09]];
    LOCAL CONST Robtarget Tr_meulage_motif_1_116 := [[-45.0666015625,178.2644375,53.5840859375],[0.205457264684473,-0.183019148705642,0.639481640238406,-0.717881978735665],[0,0,0,0],[8.999999E+09,8.999999E+09,8.999999E+09,8.999999E+09,8.999999E+09,8.999999E+09]];
    LOCAL CONST Robtarget Tr_meulage_motif_1_117 := [[-44.1784375,178.72396875,53.5840859375],[0.205457264684473,-0.183019148705642,0.639481640238406,-0.717881978735665],[0,0,0,0],[8.999999E+09,8.999999E+09,8.999999E+09,8.999999E+09,8.999999E+09,8.999999E+09]];
    LOCAL CONST Robtarget Tr_meulage_motif_1_118 := [[-43.29027734375,179.1835,53.5840859375],[0.205457264684473,-0.183019148705642,0.639481640238406,-0.717881978735665],[0,0,0,0],[8.999999E+09,8.999999E+09,8.999999E+09,8.999999E+09,8.999999E+09,8.999999E+09]];
    LOCAL CONST Robtarget Tr_meulage_motif_1_119 := [[-42.40211328125,179.643015625,53.5840859375],[0.205457264684473,-0.183019148705642,0.639481640238406,-0.717881978735665],[0,0,0,0],[8.999999E+09,8.999999E+09,8.999999E+09,8.999999E+09,8.999999E+09,8.999999E+09]];
    LOCAL CONST Robtarget Tr_meulage_motif_1_120 := [[-41.51394921875,180.102546875,53.5840859375],[0.205457264684473,-0.183019148705642,0.639481640238406,-0.717881978735665],[0,0,0,0],[8.999999E+09,8.999999E+09,8.999999E+09,8.999999E+09,8.999999E+09,8.999999E+09]];
    LOCAL CONST Robtarget Tr_meulage_motif_1_121 := [[-40.62578515625,180.562078125,53.5840859375],[0.205457264684473,-0.183019148705642,0.639481640238406,-0.717881978735665],[0,0,0,0],[8.999999E+09,8.999999E+09,8.999999E+09,8.999999E+09,8.999999E+09,8.999999E+09]];
    LOCAL CONST Robtarget Tr_meulage_motif_1_122 := [[-39.73762109375,181.021609375,53.5840859375],[0.205457264684473,-0.183019148705642,0.639481640238406,-0.717881978735665],[0,0,0,0],[8.999999E+09,8.999999E+09,8.999999E+09,8.999999E+09,8.999999E+09,8.999999E+09]];
    LOCAL CONST Robtarget Tr_meulage_motif_1_123 := [[-38.84945703125,181.481125,53.58408203125],[0.205457264684473,-0.183019148705642,0.639481640238406,-0.717881978735665],[0,0,0,0],[8.999999E+09,8.999999E+09,8.999999E+09,8.999999E+09,8.999999E+09,8.999999E+09]];
    LOCAL CONST Robtarget Tr_meulage_motif_1_124 := [[-37.96129296875,181.94065625,53.58408203125],[0.205457264684473,-0.183019148705642,0.639481640238406,-0.717881978735665],[0,0,0,0],[8.999999E+09,8.999999E+09,8.999999E+09,8.999999E+09,8.999999E+09,8.999999E+09]];
    LOCAL CONST Robtarget Tr_meulage_motif_1_125 := [[-37.07312890625,182.4001875,53.58408203125],[0.205457264684473,-0.183019148705642,0.639481640238406,-0.717881978735665],[0,0,0,0],[8.999999E+09,8.999999E+09,8.999999E+09,8.999999E+09,8.999999E+09,8.999999E+09]];
    LOCAL CONST Robtarget Tr_meulage_motif_1_126 := [[-36.18496875,182.85971875,53.58408203125],[0.205457264684473,-0.183019148705642,0.639481640238406,-0.717881978735665],[0,0,0,0],[8.999999E+09,8.999999E+09,8.999999E+09,8.999999E+09,8.999999E+09,8.999999E+09]];
    LOCAL CONST Robtarget Tr_meulage_motif_1_127 := [[-35.2968046875,183.31925,53.58408203125],[0.205457264684473,-0.183019148705642,0.639481640238406,-0.717881978735665],[0,0,0,0],[8.999999E+09,8.999999E+09,8.999999E+09,8.999999E+09,8.999999E+09,8.999999E+09]];
    LOCAL CONST Robtarget Tr_meulage_motif_1_128 := [[-34.408640625,183.778765625,53.58408203125],[0.205457264684473,-0.183019148705642,0.639481640238406,-0.717881978735665],[0,0,0,0],[8.999999E+09,8.999999E+09,8.999999E+09,8.999999E+09,8.999999E+09,8.999999E+09]];
    LOCAL CONST Robtarget Tr_meulage_motif_1_129 := [[-33.5204765625,184.238296875,53.58408203125],[0.205457264684473,-0.183019148705642,0.639481640238406,-0.717881978735665],[0,0,0,0],[8.999999E+09,8.999999E+09,8.999999E+09,8.999999E+09,8.999999E+09,8.999999E+09]];
    LOCAL CONST Robtarget Tr_meulage_motif_1_130 := [[-32.6323125,184.697828125,53.58408203125],[0.205457264684473,-0.183019148705642,0.639481640238406,-0.717881978735665],[0,0,0,0],[8.999999E+09,8.999999E+09,8.999999E+09,8.999999E+09,8.999999E+09,8.999999E+09]];
    LOCAL CONST Robtarget Tr_meulage_motif_1_131 := [[-31.7441484375,185.157359375,53.58408203125],[0.205457264684473,-0.183019148705642,0.639481640238406,-0.717881978735665],[0,0,0,0],[8.999999E+09,8.999999E+09,8.999999E+09,8.999999E+09,8.999999E+09,8.999999E+09]];
    LOCAL CONST Robtarget Tr_meulage_motif_1_132 := [[-30.855986328125,185.616875,53.584078125],[0.205457264684473,-0.183019148705642,0.639481640238406,-0.717881978735665],[0,0,0,0],[8.999999E+09,8.999999E+09,8.999999E+09,8.999999E+09,8.999999E+09,8.999999E+09]];
    LOCAL CONST Robtarget Tr_meulage_motif_1_133 := [[-29.967822265625,186.07640625,53.584078125],[0.205457264684473,-0.183019148705642,0.639481640238406,-0.717881978735665],[0,0,0,0],[8.999999E+09,8.999999E+09,8.999999E+09,8.999999E+09,8.999999E+09,8.999999E+09]];
    LOCAL CONST Robtarget Tr_meulage_motif_1_134 := [[-29.079658203125,186.5359375,53.584078125],[0.205457264684473,-0.183019148705642,0.639481640238406,-0.717881978735665],[0,0,0,0],[8.999999E+09,8.999999E+09,8.999999E+09,8.999999E+09,8.999999E+09,8.999999E+09]];
    LOCAL CONST Robtarget Tr_meulage_motif_1_135 := [[-28.191494140625,186.99546875,53.584078125],[0.205457264684473,-0.183019148705642,0.639481640238406,-0.717881978735665],[0,0,0,0],[8.999999E+09,8.999999E+09,8.999999E+09,8.999999E+09,8.999999E+09,8.999999E+09]];
    LOCAL CONST Robtarget Tr_meulage_motif_1_136 := [[-27.30333203125,187.454984375,53.584078125],[0.205457264684473,-0.183019148705642,0.639481640238406,-0.717881978735665],[0,0,0,0],[8.999999E+09,8.999999E+09,8.999999E+09,8.999999E+09,8.999999E+09,8.999999E+09]];
    LOCAL CONST Robtarget Tr_meulage_motif_1_137 := [[-26.41516796875,187.914515625,53.584078125],[0.205457264684473,-0.183019148705642,0.639481640238406,-0.717881978735665],[0,0,0,0],[8.999999E+09,8.999999E+09,8.999999E+09,8.999999E+09,8.999999E+09,8.999999E+09]];
    LOCAL CONST Robtarget Tr_meulage_motif_1_138 := [[-25.52700390625,188.374046875,53.584078125],[0.205457264684473,-0.183019148705642,0.639481640238406,-0.717881978735665],[0,0,0,0],[8.999999E+09,8.999999E+09,8.999999E+09,8.999999E+09,8.999999E+09,8.999999E+09]];
    LOCAL CONST Robtarget Tr_meulage_motif_1_139 := [[-24.63883984375,188.833578125,53.584078125],[0.205457264684473,-0.183019148705642,0.639481640238406,-0.717881978735665],[0,0,0,0],[8.999999E+09,8.999999E+09,8.999999E+09,8.999999E+09,8.999999E+09,8.999999E+09]];
    LOCAL CONST Robtarget Tr_meulage_motif_1_140 := [[-23.75067578125,189.29309375,53.58407421875],[0.205457264684473,-0.183019148705642,0.639481640238406,-0.717881978735665],[0,0,0,0],[8.999999E+09,8.999999E+09,8.999999E+09,8.999999E+09,8.999999E+09,8.999999E+09]];
    LOCAL CONST Robtarget Tr_meulage_motif_1_141 := [[-22.862513671875,189.752625,53.58407421875],[0.205457264684473,-0.183019148705642,0.639481640238406,-0.717881978735665],[0,0,0,0],[8.999999E+09,8.999999E+09,8.999999E+09,8.999999E+09,8.999999E+09,8.999999E+09]];
    LOCAL CONST Robtarget Tr_meulage_motif_1_142 := [[-21.974349609375,190.21215625,53.58407421875],[0.205457264684473,-0.183019148705642,0.639481640238406,-0.717881978735665],[0,0,0,0],[8.999999E+09,8.999999E+09,8.999999E+09,8.999999E+09,8.999999E+09,8.999999E+09]];
    LOCAL CONST Robtarget Tr_meulage_motif_1_143 := [[-21.086185546875,190.6716875,53.58407421875],[0.205457264684473,-0.183019148705642,0.639481640238406,-0.717881978735665],[0,0,0,0],[8.999999E+09,8.999999E+09,8.999999E+09,8.999999E+09,8.999999E+09,8.999999E+09]];
    LOCAL CONST Robtarget Tr_meulage_motif_1_144 := [[-20.198021484375,191.131203125,53.58407421875],[0.205457264684473,-0.183019148705642,0.639481640238406,-0.717881978735665],[0,0,0,0],[8.999999E+09,8.999999E+09,8.999999E+09,8.999999E+09,8.999999E+09,8.999999E+09]];
    LOCAL CONST Robtarget Tr_meulage_motif_1_145 := [[-19.309859375,191.590734375,53.58407421875],[0.205457264684473,-0.183019148705642,0.639481640238406,-0.717881978735665],[0,0,0,0],[8.999999E+09,8.999999E+09,8.999999E+09,8.999999E+09,8.999999E+09,8.999999E+09]];
    LOCAL CONST Robtarget Tr_meulage_motif_1_146 := [[-18.4216953125,192.050265625,53.58407421875],[0.205457264684473,-0.183019148705642,0.639481640238406,-0.717881978735665],[0,0,0,0],[8.999999E+09,8.999999E+09,8.999999E+09,8.999999E+09,8.999999E+09,8.999999E+09]];
    LOCAL CONST Robtarget Tr_meulage_motif_1_147 := [[-17.53353125,192.509796875,53.58407421875],[0.205457264684473,-0.183019148705642,0.639481640238406,-0.717881978735665],[0,0,0,0],[8.999999E+09,8.999999E+09,8.999999E+09,8.999999E+09,8.999999E+09,8.999999E+09]];
    LOCAL CONST Robtarget Tr_meulage_motif_1_148 := [[-16.6453671875,192.9693125,53.58407421875],[0.205457264684473,-0.183019148705642,0.639481640238406,-0.717881978735665],[0,0,0,0],[8.999999E+09,8.999999E+09,8.999999E+09,8.999999E+09,8.999999E+09,8.999999E+09]];
    LOCAL CONST Robtarget Tr_meulage_motif_1_149 := [[-15.7572041015625,193.42884375,53.5840703125],[0.205457264684473,-0.183019148705642,0.639481640238406,-0.717881978735665],[0,0,0,0],[8.999999E+09,8.999999E+09,8.999999E+09,8.999999E+09,8.999999E+09,8.999999E+09]];
    LOCAL CONST Robtarget Tr_meulage_motif_1_150 := [[-14.869041015625,193.888375,53.5840703125],[0.205457264684473,-0.183019148705642,0.639481640238406,-0.717881978735665],[0,0,0,0],[8.999999E+09,8.999999E+09,8.999999E+09,8.999999E+09,8.999999E+09,8.999999E+09]];
    LOCAL CONST Robtarget Tr_meulage_motif_1_151 := [[-13.9878876953125,194.345265625,53.47348046875],[0.205457264684473,-0.183019148705642,0.639481640238406,-0.717881978735665],[0,0,0,0],[8.999999E+09,8.999999E+09,8.999999E+09,8.999999E+09,8.999999E+09,8.999999E+09]];
    LOCAL CONST Robtarget Tr_meulage_motif_1_152 := [[-13.1480146484375,194.781703125,53.26230078125],[0.205457264684473,-0.183019148705642,0.639481640238406,-0.717881978735665],[0,0,0,0],[8.999999E+09,8.999999E+09,8.999999E+09,8.999999E+09,8.999999E+09,8.999999E+09]];
    LOCAL CONST Robtarget Tr_meulage_motif_1_153 := [[-12.39165625,195.17546875,52.99046484375],[0.205457264684473,-0.183019148705642,0.639481640238406,-0.717881978735665],[0,0,0,0],[8.999999E+09,8.999999E+09,8.999999E+09,8.999999E+09,8.999999E+09,8.999999E+09]];
    LOCAL CONST Robtarget Tr_meulage_motif_1_154 := [[-11.7608408203125,195.504578125,52.68631640625],[0.205457264684473,-0.183019148705642,0.639481640238406,-0.717881978735665],[0,0,0,0],[8.999999E+09,8.999999E+09,8.999999E+09,8.999999E+09,8.999999E+09,8.999999E+09]];
    LOCAL CONST Robtarget Tr_meulage_motif_1_155 := [[-10.8444892578125,195.984640625,52.0238046875],[0.205457264684473,-0.183019148705642,0.639481640238406,-0.717881978735665],[0,0,0,0],[8.999999E+09,8.999999E+09,8.999999E+09,8.999999E+09,8.999999E+09,8.999999E+09]];
    LOCAL CONST Robtarget Tr_meulage_motif_1_156 := [[-10.0467236328125,196.405484375,51.1218984375],[0.205457264684473,-0.183019148705642,0.639481640238406,-0.717881978735665],[0,0,0,0],[8.999999E+09,8.999999E+09,8.999999E+09,8.999999E+09,8.999999E+09,8.999999E+09]];
    LOCAL CONST Robtarget Tr_meulage_motif_1_157 := [[-9.5754140625,196.65871875,50.0758984375],[0.205457264684473,-0.183019148705642,0.639481640238406,-0.717881978735665],[0,0,0,0],[8.999999E+09,8.999999E+09,8.999999E+09,8.999999E+09,8.999999E+09,8.999999E+09]];
    LOCAL CONST Robtarget Tr_meulage_motif_1_158 := [[-9.4138369140625,196.74853125,49.382703125],[0.205457264684473,-0.183019148705642,0.639481640238406,-0.717881978735665],[0,0,0,0],[8.999999E+09,8.999999E+09,8.999999E+09,8.999999E+09,8.999999E+09,8.999999E+09]];
    LOCAL CONST Robtarget Tr_meulage_motif_1_159 := [[-9.3599521484375,196.7833125,48.6127265625],[0.205457264684473,-0.183019148705642,0.639481640238406,-0.717881978735665],[0,0,0,0],[8.999999E+09,8.999999E+09,8.999999E+09,8.999999E+09,8.999999E+09,8.999999E+09]];
    LOCAL CONST Robtarget Tr_meulage_motif_1_160 := [[-9.42222265625,196.758,47.842875],[0.205457264684473,-0.183019148705642,0.639481640238406,-0.717881978735665],[0,0,0,0],[8.999999E+09,8.999999E+09,8.999999E+09,8.999999E+09,8.999999E+09,8.999999E+09]];
    LOCAL CONST Robtarget Tr_meulage_motif_1_161 := [[-9.79894921875,196.57303125,46.73466015625],[0.205457264684473,-0.183019148705642,0.639481640238406,-0.717881978735665],[0,0,0,0],[8.999999E+09,8.999999E+09,8.999999E+09,8.999999E+09,8.999999E+09,8.999999E+09]];
    LOCAL CONST Robtarget Tr_meulage_motif_1_162 := [[-10.1690703125,196.386796875,46.1489921875],[0.205457264684473,-0.183019148705642,0.639481640238406,-0.717881978735665],[0,0,0,0],[8.999999E+09,8.999999E+09,8.999999E+09,8.999999E+09,8.999999E+09,8.999999E+09]];
    LOCAL CONST Robtarget Tr_meulage_motif_1_163 := [[-10.9602314453125,195.98540625,45.26189453125],[0.205457264684473,-0.183019148705642,0.639481640238406,-0.717881978735665],[0,0,0,0],[8.999999E+09,8.999999E+09,8.999999E+09,8.999999E+09,8.999999E+09,8.999999E+09]];
    LOCAL CONST Robtarget Tr_meulage_motif_1_164 := [[-11.4819345703125,195.719203125,44.84759765625],[0.205457264684473,-0.183019148705642,0.639481640238406,-0.717881978735665],[0,0,0,0],[8.999999E+09,8.999999E+09,8.999999E+09,8.999999E+09,8.999999E+09,8.999999E+09]];
    LOCAL CONST Robtarget Tr_meulage_motif_1_165 := [[-12.476810546875,195.20934375,44.30351953125],[0.205457264684473,-0.183019148705642,0.639481640238406,-0.717881978735665],[0,0,0,0],[8.999999E+09,8.999999E+09,8.999999E+09,8.999999E+09,8.999999E+09,8.999999E+09]];
    LOCAL CONST Robtarget Tr_meulage_motif_1_166 := [[-13.211154296875,194.832046875,44.00803125],[0.205457264684473,-0.183019148705642,0.639481640238406,-0.717881978735665],[0,0,0,0],[8.999999E+09,8.999999E+09,8.999999E+09,8.999999E+09,8.999999E+09,8.999999E+09]];
    LOCAL CONST Robtarget Tr_meulage_motif_1_167 := [[-14.039671875,194.40521875,43.8035703125],[0.205457264684473,-0.183019148705642,0.639481640238406,-0.717881978735665],[0,0,0,0],[8.999999E+09,8.999999E+09,8.999999E+09,8.999999E+09,8.999999E+09,8.999999E+09]];
    LOCAL CONST Robtarget Tr_meulage_motif_1_168 := [[-14.911857421875,193.9549375,43.69498046875],[0.205457264684473,-0.183019148705642,0.639481640238406,-0.717881978735665],[0,0,0,0],[8.999999E+09,8.999999E+09,8.999999E+09,8.999999E+09,8.999999E+09,8.999999E+09]];
    LOCAL CONST Robtarget Tr_meulage_motif_1_169 := [[-15.7938203125,193.499609375,43.584390625],[0.205457264684473,-0.183019148705642,0.639481640238406,-0.717881978735665],[0,0,0,0],[8.999999E+09,8.999999E+09,8.999999E+09,8.999999E+09,8.999999E+09,8.999999E+09]];
    LOCAL CONST Robtarget Tr_meulage_motif_1_170 := [[-16.681984375,193.040078125,43.584390625],[0.205457264684473,-0.183019148705642,0.639481640238406,-0.717881978735665],[0,0,0,0],[8.999999E+09,8.999999E+09,8.999999E+09,8.999999E+09,8.999999E+09,8.999999E+09]];
    LOCAL CONST Robtarget Tr_meulage_motif_1_171 := [[-17.570146484375,192.580546875,43.584390625],[0.205457264684473,-0.183019148705642,0.639481640238406,-0.717881978735665],[0,0,0,0],[8.999999E+09,8.999999E+09,8.999999E+09,8.999999E+09,8.999999E+09,8.999999E+09]];
    LOCAL CONST Robtarget Tr_meulage_motif_1_172 := [[-18.458310546875,192.121015625,43.584390625],[0.205457264684473,-0.183019148705642,0.639481640238406,-0.717881978735665],[0,0,0,0],[8.999999E+09,8.999999E+09,8.999999E+09,8.999999E+09,8.999999E+09,8.999999E+09]];
    LOCAL CONST Robtarget Tr_meulage_motif_1_173 := [[-19.346474609375,191.6615,43.584390625],[0.205457264684473,-0.183019148705642,0.639481640238406,-0.717881978735665],[0,0,0,0],[8.999999E+09,8.999999E+09,8.999999E+09,8.999999E+09,8.999999E+09,8.999999E+09]];
    LOCAL CONST Robtarget Tr_meulage_motif_1_174 := [[-20.234638671875,191.20196875,43.584390625],[0.205457264684473,-0.183019148705642,0.639481640238406,-0.717881978735665],[0,0,0,0],[8.999999E+09,8.999999E+09,8.999999E+09,8.999999E+09,8.999999E+09,8.999999E+09]];
    LOCAL CONST Robtarget Tr_meulage_motif_1_175 := [[-21.122802734375,190.7424375,43.584390625],[0.205457264684473,-0.183019148705642,0.639481640238406,-0.717881978735665],[0,0,0,0],[8.999999E+09,8.999999E+09,8.999999E+09,8.999999E+09,8.999999E+09,8.999999E+09]];
    LOCAL CONST Robtarget Tr_meulage_motif_1_176 := [[-22.01096484375,190.28290625,43.58439453125],[0.205457264684473,-0.183019148705642,0.639481640238406,-0.717881978735665],[0,0,0,0],[8.999999E+09,8.999999E+09,8.999999E+09,8.999999E+09,8.999999E+09,8.999999E+09]];
    LOCAL CONST Robtarget Tr_meulage_motif_1_177 := [[-22.89912890625,189.823390625,43.58439453125],[0.205457264684473,-0.183019148705642,0.639481640238406,-0.717881978735665],[0,0,0,0],[8.999999E+09,8.999999E+09,8.999999E+09,8.999999E+09,8.999999E+09,8.999999E+09]];
    LOCAL CONST Robtarget Tr_meulage_motif_1_178 := [[-23.78729296875,189.363859375,43.58439453125],[0.205457264684473,-0.183019148705642,0.639481640238406,-0.717881978735665],[0,0,0,0],[8.999999E+09,8.999999E+09,8.999999E+09,8.999999E+09,8.999999E+09,8.999999E+09]];
    LOCAL CONST Robtarget Tr_meulage_motif_1_179 := [[-24.67545703125,188.904328125,43.58439453125],[0.205457264684473,-0.183019148705642,0.639481640238406,-0.717881978735665],[0,0,0,0],[8.999999E+09,8.999999E+09,8.999999E+09,8.999999E+09,8.999999E+09,8.999999E+09]];
    LOCAL CONST Robtarget Tr_meulage_motif_1_180 := [[-25.563619140625,188.444796875,43.58439453125],[0.205457264684473,-0.183019148705642,0.639481640238406,-0.717881978735665],[0,0,0,0],[8.999999E+09,8.999999E+09,8.999999E+09,8.999999E+09,8.999999E+09,8.999999E+09]];
    LOCAL CONST Robtarget Tr_meulage_motif_1_181 := [[-26.451783203125,187.98528125,43.58439453125],[0.205457264684473,-0.183019148705642,0.639481640238406,-0.717881978735665],[0,0,0,0],[8.999999E+09,8.999999E+09,8.999999E+09,8.999999E+09,8.999999E+09,8.999999E+09]];
    LOCAL CONST Robtarget Tr_meulage_motif_1_182 := [[-27.339947265625,187.52575,43.58439453125],[0.205457264684473,-0.183019148705642,0.639481640238406,-0.717881978735665],[0,0,0,0],[8.999999E+09,8.999999E+09,8.999999E+09,8.999999E+09,8.999999E+09,8.999999E+09]];
    LOCAL CONST Robtarget Tr_meulage_motif_1_183 := [[-28.228111328125,187.06621875,43.58439453125],[0.205457264684473,-0.183019148705642,0.639481640238406,-0.717881978735665],[0,0,0,0],[8.999999E+09,8.999999E+09,8.999999E+09,8.999999E+09,8.999999E+09,8.999999E+09]];
    LOCAL CONST Robtarget Tr_meulage_motif_1_184 := [[-29.1162734375,186.6066875,43.58439453125],[0.205457264684473,-0.183019148705642,0.639481640238406,-0.717881978735665],[0,0,0,0],[8.999999E+09,8.999999E+09,8.999999E+09,8.999999E+09,8.999999E+09,8.999999E+09]];
    LOCAL CONST Robtarget Tr_meulage_motif_1_185 := [[-30.0044375,186.147171875,43.5843984375],[0.205457264684473,-0.183019148705642,0.639481640238406,-0.717881978735665],[0,0,0,0],[8.999999E+09,8.999999E+09,8.999999E+09,8.999999E+09,8.999999E+09,8.999999E+09]];
    LOCAL CONST Robtarget Tr_meulage_motif_1_186 := [[-30.8926015625,185.687640625,43.5843984375],[0.205457264684473,-0.183019148705642,0.639481640238406,-0.717881978735665],[0,0,0,0],[8.999999E+09,8.999999E+09,8.999999E+09,8.999999E+09,8.999999E+09,8.999999E+09]];
    LOCAL CONST Robtarget Tr_meulage_motif_1_187 := [[-31.780765625,185.228109375,43.5843984375],[0.205457264684473,-0.183019148705642,0.639481640238406,-0.717881978735665],[0,0,0,0],[8.999999E+09,8.999999E+09,8.999999E+09,8.999999E+09,8.999999E+09,8.999999E+09]];
    LOCAL CONST Robtarget Tr_meulage_motif_1_188 := [[-32.668927734375,184.768578125,43.5843984375],[0.205457264684473,-0.183019148705642,0.639481640238406,-0.717881978735665],[0,0,0,0],[8.999999E+09,8.999999E+09,8.999999E+09,8.999999E+09,8.999999E+09,8.999999E+09]];
    LOCAL CONST Robtarget Tr_meulage_motif_1_189 := [[-33.55709375,184.3090625,43.5843984375],[0.205457264684473,-0.183019148705642,0.639481640238406,-0.717881978735665],[0,0,0,0],[8.999999E+09,8.999999E+09,8.999999E+09,8.999999E+09,8.999999E+09,8.999999E+09]];
    LOCAL CONST Robtarget Tr_meulage_motif_1_190 := [[-34.44525390625,183.84953125,43.5843984375],[0.205457264684473,-0.183019148705642,0.639481640238406,-0.717881978735665],[0,0,0,0],[8.999999E+09,8.999999E+09,8.999999E+09,8.999999E+09,8.999999E+09,8.999999E+09]];
    LOCAL CONST Robtarget Tr_meulage_motif_1_191 := [[-35.33341796875,183.39,43.5843984375],[0.205457264684473,-0.183019148705642,0.639481640238406,-0.717881978735665],[0,0,0,0],[8.999999E+09,8.999999E+09,8.999999E+09,8.999999E+09,8.999999E+09,8.999999E+09]];
    LOCAL CONST Robtarget Tr_meulage_motif_1_192 := [[-36.22158203125,182.93046875,43.5843984375],[0.205457264684473,-0.183019148705642,0.639481640238406,-0.717881978735665],[0,0,0,0],[8.999999E+09,8.999999E+09,8.999999E+09,8.999999E+09,8.999999E+09,8.999999E+09]];
    LOCAL CONST Robtarget Tr_meulage_motif_1_193 := [[-37.10974609375,182.470953125,43.58440234375],[0.205457264684473,-0.183019148705642,0.639481640238406,-0.717881978735665],[0,0,0,0],[8.999999E+09,8.999999E+09,8.999999E+09,8.999999E+09,8.999999E+09,8.999999E+09]];
    LOCAL CONST Robtarget Tr_meulage_motif_1_194 := [[-37.99791015625,182.011421875,43.58440234375],[0.205457264684473,-0.183019148705642,0.639481640238406,-0.717881978735665],[0,0,0,0],[8.999999E+09,8.999999E+09,8.999999E+09,8.999999E+09,8.999999E+09,8.999999E+09]];
    LOCAL CONST Robtarget Tr_meulage_motif_1_195 := [[-38.88607421875,181.551890625,43.58440234375],[0.205457264684473,-0.183019148705642,0.639481640238406,-0.717881978735665],[0,0,0,0],[8.999999E+09,8.999999E+09,8.999999E+09,8.999999E+09,8.999999E+09,8.999999E+09]];
    LOCAL CONST Robtarget Tr_meulage_motif_1_196 := [[-39.77423828125,181.092359375,43.58440234375],[0.205457264684473,-0.183019148705642,0.639481640238406,-0.717881978735665],[0,0,0,0],[8.999999E+09,8.999999E+09,8.999999E+09,8.999999E+09,8.999999E+09,8.999999E+09]];
    LOCAL CONST Robtarget Tr_meulage_motif_1_197 := [[-40.66240234375,180.63284375,43.58440234375],[0.205457264684473,-0.183019148705642,0.639481640238406,-0.717881978735665],[0,0,0,0],[8.999999E+09,8.999999E+09,8.999999E+09,8.999999E+09,8.999999E+09,8.999999E+09]];
    LOCAL CONST Robtarget Tr_meulage_motif_1_198 := [[-41.55056640625,180.1733125,43.58440234375],[0.205457264684473,-0.183019148705642,0.639481640238406,-0.717881978735665],[0,0,0,0],[8.999999E+09,8.999999E+09,8.999999E+09,8.999999E+09,8.999999E+09,8.999999E+09]];
    LOCAL CONST Robtarget Tr_meulage_motif_1_199 := [[-42.4387265625,179.71378125,43.58440234375],[0.205457264684473,-0.183019148705642,0.639481640238406,-0.717881978735665],[0,0,0,0],[8.999999E+09,8.999999E+09,8.999999E+09,8.999999E+09,8.999999E+09,8.999999E+09]];
    LOCAL CONST Robtarget Tr_meulage_motif_1_200 := [[-43.326890625,179.25425,43.58440234375],[0.205457264684473,-0.183019148705642,0.639481640238406,-0.717881978735665],[0,0,0,0],[8.999999E+09,8.999999E+09,8.999999E+09,8.999999E+09,8.999999E+09,8.999999E+09]];
    LOCAL CONST Robtarget Tr_meulage_motif_1_201 := [[-44.2150546875,178.794734375,43.58440234375],[0.205457264684473,-0.183019148705642,0.639481640238406,-0.717881978735665],[0,0,0,0],[8.999999E+09,8.999999E+09,8.999999E+09,8.999999E+09,8.999999E+09,8.999999E+09]];
    LOCAL CONST Robtarget Tr_meulage_motif_1_202 := [[-45.10321875,178.335203125,43.58440625],[0.205457264684473,-0.183019148705642,0.639481640238406,-0.717881978735665],[0,0,0,0],[8.999999E+09,8.999999E+09,8.999999E+09,8.999999E+09,8.999999E+09,8.999999E+09]];
    LOCAL CONST Robtarget Tr_meulage_motif_1_203 := [[-45.9913828125,177.875671875,43.58440625],[0.205457264684473,-0.183019148705642,0.639481640238406,-0.717881978735665],[0,0,0,0],[8.999999E+09,8.999999E+09,8.999999E+09,8.999999E+09,8.999999E+09,8.999999E+09]];
    LOCAL CONST Robtarget Tr_meulage_motif_1_204 := [[-46.879546875,177.416140625,43.58440625],[0.205457264684473,-0.183019148705642,0.639481640238406,-0.717881978735665],[0,0,0,0],[8.999999E+09,8.999999E+09,8.999999E+09,8.999999E+09,8.999999E+09,8.999999E+09]];
    LOCAL CONST Robtarget Tr_meulage_motif_1_205 := [[-47.7677109375,176.956625,43.58440625],[0.205457264684473,-0.183019148705642,0.639481640238406,-0.717881978735665],[0,0,0,0],[8.999999E+09,8.999999E+09,8.999999E+09,8.999999E+09,8.999999E+09,8.999999E+09]];
    LOCAL CONST Robtarget Tr_meulage_motif_1_206 := [[-48.655875,176.49709375,43.58440625],[0.205457264684473,-0.183019148705642,0.639481640238406,-0.717881978735665],[0,0,0,0],[8.999999E+09,8.999999E+09,8.999999E+09,8.999999E+09,8.999999E+09,8.999999E+09]];
    LOCAL CONST Robtarget Tr_meulage_motif_1_207 := [[-49.54403515625,176.0375625,43.58440625],[0.205457264684473,-0.183019148705642,0.639481640238406,-0.717881978735665],[0,0,0,0],[8.999999E+09,8.999999E+09,8.999999E+09,8.999999E+09,8.999999E+09,8.999999E+09]];
    LOCAL CONST Robtarget Tr_meulage_motif_1_208 := [[-50.43219921875,175.57803125,43.58440625],[0.205457264684473,-0.183019148705642,0.639481640238406,-0.717881978735665],[0,0,0,0],[8.999999E+09,8.999999E+09,8.999999E+09,8.999999E+09,8.999999E+09,8.999999E+09]];
    LOCAL CONST Robtarget Tr_meulage_motif_1_209 := [[-51.32036328125,175.118515625,43.58440625],[0.205457264684473,-0.183019148705642,0.639481640238406,-0.717881978735665],[0,0,0,0],[8.999999E+09,8.999999E+09,8.999999E+09,8.999999E+09,8.999999E+09,8.999999E+09]];
    LOCAL CONST Robtarget Tr_meulage_motif_1_210 := [[-52.20852734375,174.658984375,43.58440625],[0.205457264684473,-0.183019148705642,0.639481640238406,-0.717881978735665],[0,0,0,0],[8.999999E+09,8.999999E+09,8.999999E+09,8.999999E+09,8.999999E+09,8.999999E+09]];
    LOCAL CONST Robtarget Tr_meulage_motif_1_211 := [[-53.09669140625,174.199453125,43.58441015625],[0.205457264684473,-0.183019148705642,0.639481640238406,-0.717881978735665],[0,0,0,0],[8.999999E+09,8.999999E+09,8.999999E+09,8.999999E+09,8.999999E+09,8.999999E+09]];
    LOCAL CONST Robtarget Tr_meulage_motif_1_212 := [[-53.98485546875,173.739921875,43.58441015625],[0.205457264684473,-0.183019148705642,0.639481640238406,-0.717881978735665],[0,0,0,0],[8.999999E+09,8.999999E+09,8.999999E+09,8.999999E+09,8.999999E+09,8.999999E+09]];
    LOCAL CONST Robtarget Tr_meulage_motif_1_213 := [[-54.87301953125,173.28040625,43.58441015625],[0.205457264684473,-0.183019148705642,0.639481640238406,-0.717881978735665],[0,0,0,0],[8.999999E+09,8.999999E+09,8.999999E+09,8.999999E+09,8.999999E+09,8.999999E+09]];
    LOCAL CONST Robtarget Tr_meulage_motif_1_214 := [[-55.76118359375,172.820875,43.58441015625],[0.205457264684473,-0.183019148705642,0.639481640238406,-0.717881978735665],[0,0,0,0],[8.999999E+09,8.999999E+09,8.999999E+09,8.999999E+09,8.999999E+09,8.999999E+09]];
    LOCAL CONST Robtarget Tr_meulage_motif_1_215 := [[-56.64934375,172.36134375,43.58441015625],[0.205457264684473,-0.183019148705642,0.639481640238406,-0.717881978735665],[0,0,0,0],[8.999999E+09,8.999999E+09,8.999999E+09,8.999999E+09,8.999999E+09,8.999999E+09]];
    LOCAL CONST Robtarget Tr_meulage_motif_1_216 := [[-57.5375078125,171.9018125,43.58441015625],[0.205457264684473,-0.183019148705642,0.639481640238406,-0.717881978735665],[0,0,0,0],[8.999999E+09,8.999999E+09,8.999999E+09,8.999999E+09,8.999999E+09,8.999999E+09]];
    LOCAL CONST Robtarget Tr_meulage_motif_1_217 := [[-58.425671875,171.442296875,43.58441015625],[0.205457264684473,-0.183019148705642,0.639481640238406,-0.717881978735665],[0,0,0,0],[8.999999E+09,8.999999E+09,8.999999E+09,8.999999E+09,8.999999E+09,8.999999E+09]];
    LOCAL CONST Robtarget Tr_meulage_motif_1_218 := [[-59.3138359375,170.982765625,43.58441015625],[0.205457264684473,-0.183019148705642,0.639481640238406,-0.717881978735665],[0,0,0,0],[8.999999E+09,8.999999E+09,8.999999E+09,8.999999E+09,8.999999E+09,8.999999E+09]];
    LOCAL CONST Robtarget Tr_meulage_motif_1_219 := [[-60.202,170.523234375,43.5844140625],[0.205457264684473,-0.183019148705642,0.639481640238406,-0.717881978735665],[0,0,0,0],[8.999999E+09,8.999999E+09,8.999999E+09,8.999999E+09,8.999999E+09,8.999999E+09]];
    LOCAL CONST Robtarget Tr_meulage_motif_1_220 := [[-61.0901640625,170.063703125,43.5844140625],[0.205457264684473,-0.183019148705642,0.639481640238406,-0.717881978735665],[0,0,0,0],[8.999999E+09,8.999999E+09,8.999999E+09,8.999999E+09,8.999999E+09,8.999999E+09]];
    LOCAL CONST Robtarget Tr_meulage_motif_1_221 := [[-61.978328125,169.6041875,43.5844140625],[0.205457264684473,-0.183019148705642,0.639481640238406,-0.717881978735665],[0,0,0,0],[8.999999E+09,8.999999E+09,8.999999E+09,8.999999E+09,8.999999E+09,8.999999E+09]];
    LOCAL CONST Robtarget Tr_meulage_motif_1_222 := [[-62.8664921875,169.14465625,43.5844140625],[0.205457264684473,-0.183019148705642,0.639481640238406,-0.717881978735665],[0,0,0,0],[8.999999E+09,8.999999E+09,8.999999E+09,8.999999E+09,8.999999E+09,8.999999E+09]];
    LOCAL CONST Robtarget Tr_meulage_motif_1_223 := [[-63.75465625,168.685125,43.5844140625],[0.205457264684473,-0.183019148705642,0.639481640238406,-0.717881978735665],[0,0,0,0],[8.999999E+09,8.999999E+09,8.999999E+09,8.999999E+09,8.999999E+09,8.999999E+09]];
    LOCAL CONST Robtarget Tr_meulage_motif_1_224 := [[-64.64281640625,168.22559375,43.5844140625],[0.205457264684473,-0.183019148705642,0.639481640238406,-0.717881978735665],[0,0,0,0],[8.999999E+09,8.999999E+09,8.999999E+09,8.999999E+09,8.999999E+09,8.999999E+09]];
    LOCAL CONST Robtarget Tr_meulage_motif_1_225 := [[-65.53098046875,167.766078125,43.5844140625],[0.205457264684473,-0.183019148705642,0.639481640238406,-0.717881978735665],[0,0,0,0],[8.999999E+09,8.999999E+09,8.999999E+09,8.999999E+09,8.999999E+09,8.999999E+09]];
    LOCAL CONST Robtarget Tr_meulage_motif_1_226 := [[-66.4191484375,167.306546875,43.5844140625],[0.205457264684473,-0.183019148705642,0.639481640238406,-0.717881978735665],[0,0,0,0],[8.999999E+09,8.999999E+09,8.999999E+09,8.999999E+09,8.999999E+09,8.999999E+09]];
    LOCAL CONST Robtarget Tr_meulage_motif_1_227 := [[-67.3073125,166.847015625,43.5844140625],[0.205457264684473,-0.183019148705642,0.639481640238406,-0.717881978735665],[0,0,0,0],[8.999999E+09,8.999999E+09,8.999999E+09,8.999999E+09,8.999999E+09,8.999999E+09]];
    LOCAL CONST Robtarget Tr_meulage_motif_1_228 := [[-68.19546875,166.387484375,43.58441796875],[0.205457264684473,-0.183019148705642,0.639481640238406,-0.717881978735665],[0,0,0,0],[8.999999E+09,8.999999E+09,8.999999E+09,8.999999E+09,8.999999E+09,8.999999E+09]];
    LOCAL CONST Robtarget Tr_meulage_motif_1_229 := [[-69.0836328125,165.92796875,43.58441796875],[0.205457264684473,-0.183019148705642,0.639481640238406,-0.717881978735665],[0,0,0,0],[8.999999E+09,8.999999E+09,8.999999E+09,8.999999E+09,8.999999E+09,8.999999E+09]];
    LOCAL CONST Robtarget Tr_meulage_motif_1_230 := [[-69.971796875,165.4684375,43.58441796875],[0.205457264684473,-0.183019148705642,0.639481640238406,-0.717881978735665],[0,0,0,0],[8.999999E+09,8.999999E+09,8.999999E+09,8.999999E+09,8.999999E+09,8.999999E+09]];
    LOCAL CONST Robtarget Tr_meulage_motif_1_231 := [[-70.853765625,165.013109375,43.473828125],[0.205457264684473,-0.183019148705642,0.639481640238406,-0.717881978735665],[0,0,0,0],[8.999999E+09,8.999999E+09,8.999999E+09,8.999999E+09,8.999999E+09,8.999999E+09]];
    LOCAL CONST Robtarget Tr_meulage_motif_1_232 := [[-71.6951796875,164.57965625,43.2626484375],[0.205457264684473,-0.183019148705642,0.639481640238406,-0.717881978735665],[0,0,0,0],[8.999999E+09,8.999999E+09,8.999999E+09,8.999999E+09,8.999999E+09,8.999999E+09]];
    LOCAL CONST Robtarget Tr_meulage_motif_1_233 := [[-72.45353125,164.189734375,42.9908125],[0.205457264684473,-0.183019148705642,0.639481640238406,-0.717881978735665],[0,0,0,0],[8.999999E+09,8.999999E+09,8.999999E+09,8.999999E+09,8.999999E+09,8.999999E+09]];
    LOCAL CONST Robtarget Tr_meulage_motif_1_234 := [[-73.120578125,163.847078125,42.7148828125],[0.205457264684473,-0.183019148705642,0.639481640238406,-0.717881978735665],[0,0,0,0],[8.999999E+09,8.999999E+09,8.999999E+09,8.999999E+09,8.999999E+09,8.999999E+09]];
    LOCAL CONST Robtarget Tr_meulage_motif_1_235 := [[-74.1007890625,163.34546875,42.09877734375],[0.205457264684473,-0.183019148705642,0.639481640238406,-0.717881978735665],[0,0,0,0],[8.999999E+09,8.999999E+09,8.999999E+09,8.999999E+09,8.999999E+09,8.999999E+09]];
    LOCAL CONST Robtarget Tr_meulage_motif_1_236 := [[-75.0132578125,162.88096875,41.2511484375],[0.205457264684473,-0.183019148705642,0.639481640238406,-0.717881978735665],[0,0,0,0],[8.999999E+09,8.999999E+09,8.999999E+09,8.999999E+09,8.999999E+09,8.999999E+09]];
    LOCAL CONST Robtarget Tr_meulage_motif_1_237 := [[-75.7698671875,162.4986875,40.22730859375],[0.205457264684473,-0.183019148705642,0.639481640238406,-0.717881978735665],[0,0,0,0],[8.999999E+09,8.999999E+09,8.999999E+09,8.999999E+09,8.999999E+09,8.999999E+09]];
    LOCAL CONST Robtarget Tr_meulage_motif_1_238 := [[-76.207515625,162.282265625,39.11115625],[0.205457264684473,-0.183019148705642,0.639481640238406,-0.717881978735665],[0,0,0,0],[8.999999E+09,8.999999E+09,8.999999E+09,8.999999E+09,8.999999E+09,8.999999E+09]];
    LOCAL CONST Robtarget Tr_meulage_motif_1_239 := [[-76.2341015625,162.27475,38.4152109375],[0.205457264684473,-0.183019148705642,0.639481640238406,-0.717881978735665],[0,0,0,0],[8.999999E+09,8.999999E+09,8.999999E+09,8.999999E+09,8.999999E+09,8.999999E+09]];
    LOCAL CONST Robtarget Tr_meulage_motif_1_240 := [[-76.2365234375,162.2794375,37.75398046875],[0.205457264684473,-0.183019148705642,0.639481640238406,-0.717881978735665],[0,0,0,0],[8.999999E+09,8.999999E+09,8.999999E+09,8.999999E+09,8.999999E+09,8.999999E+09]];
    LOCAL CONST Robtarget Tr_meulage_motif_1_241 := [[-76.190203125,162.309328125,37.09290625],[0.205457264684473,-0.183019148705642,0.639481640238406,-0.717881978735665],[0,0,0,0],[8.999999E+09,8.999999E+09,8.999999E+09,8.999999E+09,8.999999E+09,8.999999E+09]];
    LOCAL CONST Robtarget Tr_meulage_motif_1_242 := [[-75.7517421875,162.5460625,35.99119140625],[0.205457264684473,-0.183019148705642,0.639481640238406,-0.717881978735665],[0,0,0,0],[8.999999E+09,8.999999E+09,8.999999E+09,8.999999E+09,8.999999E+09,8.999999E+09]];
    LOCAL CONST Robtarget Tr_meulage_motif_1_243 := [[-74.9946015625,162.946828125,34.98459765625],[0.205457264684473,-0.183019148705642,0.639481640238406,-0.717881978735665],[0,0,0,0],[8.999999E+09,8.999999E+09,8.999999E+09,8.999999E+09,8.999999E+09,8.999999E+09]];
    LOCAL CONST Robtarget Tr_meulage_motif_1_244 := [[-74.08865625,163.423,34.15575],[0.205457264684473,-0.183019148705642,0.639481640238406,-0.717881978735665],[0,0,0,0],[8.999999E+09,8.999999E+09,8.999999E+09,8.999999E+09,8.999999E+09,8.999999E+09]];
    LOCAL CONST Robtarget Tr_meulage_motif_1_245 := [[-73.4798828125,163.741515625,33.76001171875],[0.205457264684473,-0.183019148705642,0.639481640238406,-0.717881978735665],[0,0,0,0],[8.999999E+09,8.999999E+09,8.999999E+09,8.999999E+09,8.999999E+09,8.999999E+09]];
    LOCAL CONST Robtarget Tr_meulage_motif_1_246 := [[-72.4530390625,164.277171875,33.27249609375],[0.205457264684473,-0.183019148705642,0.639481640238406,-0.717881978735665],[0,0,0,0],[8.999999E+09,8.999999E+09,8.999999E+09,8.999999E+09,8.999999E+09,8.999999E+09]];
    LOCAL CONST Robtarget Tr_meulage_motif_1_247 := [[-71.7034765625,164.667359375,33.00841015625],[0.205457264684473,-0.183019148705642,0.639481640238406,-0.717881978735665],[0,0,0,0],[8.999999E+09,8.999999E+09,8.999999E+09,8.999999E+09,8.999999E+09,8.999999E+09]];
    LOCAL CONST Robtarget Tr_meulage_motif_1_248 := [[-70.876453125,165.097078125,32.80394921875],[0.205457264684473,-0.183019148705642,0.639481640238406,-0.717881978735665],[0,0,0,0],[8.999999E+09,8.999999E+09,8.999999E+09,8.999999E+09,8.999999E+09,8.999999E+09]];
    LOCAL CONST Robtarget Tr_meulage_motif_1_249 := [[-70.0050703125,165.54890625,32.695357421875],[0.205457264684473,-0.183019148705642,0.639481640238406,-0.717881978735665],[0,0,0,0],[8.999999E+09,8.999999E+09,8.999999E+09,8.999999E+09,8.999999E+09,8.999999E+09]];
    LOCAL CONST Robtarget Tr_meulage_motif_1_250 := [[-69.1239140625,166.005796875,32.584765625],[0.205457264684473,-0.183019148705642,0.639481640238406,-0.717881978735665],[0,0,0,0],[8.999999E+09,8.999999E+09,8.999999E+09,8.999999E+09,8.999999E+09,8.999999E+09]];
    LOCAL CONST Robtarget Tr_meulage_motif_1_251 := [[-68.23575,166.465328125,32.584765625],[0.205457264684473,-0.183019148705642,0.639481640238406,-0.717881978735665],[0,0,0,0],[8.999999E+09,8.999999E+09,8.999999E+09,8.999999E+09,8.999999E+09,8.999999E+09]];
    LOCAL CONST Robtarget Tr_meulage_motif_1_252 := [[-67.3475859375,166.924859375,32.584765625],[0.205457264684473,-0.183019148705642,0.639481640238406,-0.717881978735665],[0,0,0,0],[8.999999E+09,8.999999E+09,8.999999E+09,8.999999E+09,8.999999E+09,8.999999E+09]];
    LOCAL CONST Robtarget Tr_meulage_motif_1_253 := [[-66.459421875,167.384375,32.584763671875],[0.205457264684473,-0.183019148705642,0.639481640238406,-0.717881978735665],[0,0,0,0],[8.999999E+09,8.999999E+09,8.999999E+09,8.999999E+09,8.999999E+09,8.999999E+09]];
    LOCAL CONST Robtarget Tr_meulage_motif_1_254 := [[-65.5712578125,167.84390625,32.584763671875],[0.205457264684473,-0.183019148705642,0.639481640238406,-0.717881978735665],[0,0,0,0],[8.999999E+09,8.999999E+09,8.999999E+09,8.999999E+09,8.999999E+09,8.999999E+09]];
    LOCAL CONST Robtarget Tr_meulage_motif_1_255 := [[-64.68309375,168.3034375,32.584763671875],[0.205457264684473,-0.183019148705642,0.639481640238406,-0.717881978735665],[0,0,0,0],[8.999999E+09,8.999999E+09,8.999999E+09,8.999999E+09,8.999999E+09,8.999999E+09]];
    LOCAL CONST Robtarget Tr_meulage_motif_1_256 := [[-63.79493359375,168.76296875,32.584763671875],[0.205457264684473,-0.183019148705642,0.639481640238406,-0.717881978735665],[0,0,0,0],[8.999999E+09,8.999999E+09,8.999999E+09,8.999999E+09,8.999999E+09,8.999999E+09]];
    LOCAL CONST Robtarget Tr_meulage_motif_1_257 := [[-62.90676953125,169.222484375,32.584763671875],[0.205457264684473,-0.183019148705642,0.639481640238406,-0.717881978735665],[0,0,0,0],[8.999999E+09,8.999999E+09,8.999999E+09,8.999999E+09,8.999999E+09,8.999999E+09]];
    LOCAL CONST Robtarget Tr_meulage_motif_1_258 := [[-62.01860546875,169.682015625,32.58476171875],[0.205457264684473,-0.183019148705642,0.639481640238406,-0.717881978735665],[0,0,0,0],[8.999999E+09,8.999999E+09,8.999999E+09,8.999999E+09,8.999999E+09,8.999999E+09]];
    LOCAL CONST Robtarget Tr_meulage_motif_1_259 := [[-61.13044140625,170.141546875,32.58476171875],[0.205457264684473,-0.183019148705642,0.639481640238406,-0.717881978735665],[0,0,0,0],[8.999999E+09,8.999999E+09,8.999999E+09,8.999999E+09,8.999999E+09,8.999999E+09]];
    LOCAL CONST Robtarget Tr_meulage_motif_1_260 := [[-60.24227734375,170.601078125,32.58476171875],[0.205457264684473,-0.183019148705642,0.639481640238406,-0.717881978735665],[0,0,0,0],[8.999999E+09,8.999999E+09,8.999999E+09,8.999999E+09,8.999999E+09,8.999999E+09]];
    LOCAL CONST Robtarget Tr_meulage_motif_1_261 := [[-59.35411328125,171.06059375,32.58476171875],[0.205457264684473,-0.183019148705642,0.639481640238406,-0.717881978735665],[0,0,0,0],[8.999999E+09,8.999999E+09,8.999999E+09,8.999999E+09,8.999999E+09,8.999999E+09]];
    LOCAL CONST Robtarget Tr_meulage_motif_1_262 := [[-58.46594921875,171.520125,32.584759765625],[0.205457264684473,-0.183019148705642,0.639481640238406,-0.717881978735665],[0,0,0,0],[8.999999E+09,8.999999E+09,8.999999E+09,8.999999E+09,8.999999E+09,8.999999E+09]];
    LOCAL CONST Robtarget Tr_meulage_motif_1_263 := [[-57.57778515625,171.97965625,32.584759765625],[0.205457264684473,-0.183019148705642,0.639481640238406,-0.717881978735665],[0,0,0,0],[8.999999E+09,8.999999E+09,8.999999E+09,8.999999E+09,8.999999E+09,8.999999E+09]];
    LOCAL CONST Robtarget Tr_meulage_motif_1_264 := [[-56.689625,172.4391875,32.584759765625],[0.205457264684473,-0.183019148705642,0.639481640238406,-0.717881978735665],[0,0,0,0],[8.999999E+09,8.999999E+09,8.999999E+09,8.999999E+09,8.999999E+09,8.999999E+09]];
    LOCAL CONST Robtarget Tr_meulage_motif_1_265 := [[-55.8014609375,172.898703125,32.584759765625],[0.205457264684473,-0.183019148705642,0.639481640238406,-0.717881978735665],[0,0,0,0],[8.999999E+09,8.999999E+09,8.999999E+09,8.999999E+09,8.999999E+09,8.999999E+09]];
    LOCAL CONST Robtarget Tr_meulage_motif_1_266 := [[-54.913296875,173.358234375,32.5847578125],[0.205457264684473,-0.183019148705642,0.639481640238406,-0.717881978735665],[0,0,0,0],[8.999999E+09,8.999999E+09,8.999999E+09,8.999999E+09,8.999999E+09,8.999999E+09]];
    LOCAL CONST Robtarget Tr_meulage_motif_1_267 := [[-54.0251328125,173.817765625,32.5847578125],[0.205457264684473,-0.183019148705642,0.639481640238406,-0.717881978735665],[0,0,0,0],[8.999999E+09,8.999999E+09,8.999999E+09,8.999999E+09,8.999999E+09,8.999999E+09]];
    LOCAL CONST Robtarget Tr_meulage_motif_1_268 := [[-53.13696875,174.277296875,32.5847578125],[0.205457264684473,-0.183019148705642,0.639481640238406,-0.717881978735665],[0,0,0,0],[8.999999E+09,8.999999E+09,8.999999E+09,8.999999E+09,8.999999E+09,8.999999E+09]];
    LOCAL CONST Robtarget Tr_meulage_motif_1_269 := [[-52.2488046875,174.7368125,32.5847578125],[0.205457264684473,-0.183019148705642,0.639481640238406,-0.717881978735665],[0,0,0,0],[8.999999E+09,8.999999E+09,8.999999E+09,8.999999E+09,8.999999E+09,8.999999E+09]];
    LOCAL CONST Robtarget Tr_meulage_motif_1_270 := [[-51.360640625,175.19634375,32.584755859375],[0.205457264684473,-0.183019148705642,0.639481640238406,-0.717881978735665],[0,0,0,0],[8.999999E+09,8.999999E+09,8.999999E+09,8.999999E+09,8.999999E+09,8.999999E+09]];
    LOCAL CONST Robtarget Tr_meulage_motif_1_271 := [[-50.4724765625,175.655875,32.584755859375],[0.205457264684473,-0.183019148705642,0.639481640238406,-0.717881978735665],[0,0,0,0],[8.999999E+09,8.999999E+09,8.999999E+09,8.999999E+09,8.999999E+09,8.999999E+09]];
    LOCAL CONST Robtarget Tr_meulage_motif_1_272 := [[-49.5843125,176.11540625,32.584755859375],[0.205457264684473,-0.183019148705642,0.639481640238406,-0.717881978735665],[0,0,0,0],[8.999999E+09,8.999999E+09,8.999999E+09,8.999999E+09,8.999999E+09,8.999999E+09]];
    LOCAL CONST Robtarget Tr_meulage_motif_1_273 := [[-48.69615234375,176.574921875,32.584755859375],[0.205457264684473,-0.183019148705642,0.639481640238406,-0.717881978735665],[0,0,0,0],[8.999999E+09,8.999999E+09,8.999999E+09,8.999999E+09,8.999999E+09,8.999999E+09]];
    LOCAL CONST Robtarget Tr_meulage_motif_1_274 := [[-47.80798828125,177.034453125,32.584755859375],[0.205457264684473,-0.183019148705642,0.639481640238406,-0.717881978735665],[0,0,0,0],[8.999999E+09,8.999999E+09,8.999999E+09,8.999999E+09,8.999999E+09,8.999999E+09]];
    LOCAL CONST Robtarget Tr_meulage_motif_1_275 := [[-46.91982421875,177.493984375,32.58475390625],[0.205457264684473,-0.183019148705642,0.639481640238406,-0.717881978735665],[0,0,0,0],[8.999999E+09,8.999999E+09,8.999999E+09,8.999999E+09,8.999999E+09,8.999999E+09]];
    LOCAL CONST Robtarget Tr_meulage_motif_1_276 := [[-46.03166015625,177.953515625,32.58475390625],[0.205457264684473,-0.183019148705642,0.639481640238406,-0.717881978735665],[0,0,0,0],[8.999999E+09,8.999999E+09,8.999999E+09,8.999999E+09,8.999999E+09,8.999999E+09]];
    LOCAL CONST Robtarget Tr_meulage_motif_1_277 := [[-45.14349609375,178.41303125,32.58475390625],[0.205457264684473,-0.183019148705642,0.639481640238406,-0.717881978735665],[0,0,0,0],[8.999999E+09,8.999999E+09,8.999999E+09,8.999999E+09,8.999999E+09,8.999999E+09]];
    LOCAL CONST Robtarget Tr_meulage_motif_1_278 := [[-44.25533203125,178.8725625,32.58475390625],[0.205457264684473,-0.183019148705642,0.639481640238406,-0.717881978735665],[0,0,0,0],[8.999999E+09,8.999999E+09,8.999999E+09,8.999999E+09,8.999999E+09,8.999999E+09]];
    LOCAL CONST Robtarget Tr_meulage_motif_1_279 := [[-43.36716796875,179.33209375,32.584751953125],[0.205457264684473,-0.183019148705642,0.639481640238406,-0.717881978735665],[0,0,0,0],[8.999999E+09,8.999999E+09,8.999999E+09,8.999999E+09,8.999999E+09,8.999999E+09]];
    LOCAL CONST Robtarget Tr_meulage_motif_1_280 := [[-42.47900390625,179.791625,32.584751953125],[0.205457264684473,-0.183019148705642,0.639481640238406,-0.717881978735665],[0,0,0,0],[8.999999E+09,8.999999E+09,8.999999E+09,8.999999E+09,8.999999E+09,8.999999E+09]];
    LOCAL CONST Robtarget Tr_meulage_motif_1_281 := [[-41.59084375,180.251140625,32.584751953125],[0.205457264684473,-0.183019148705642,0.639481640238406,-0.717881978735665],[0,0,0,0],[8.999999E+09,8.999999E+09,8.999999E+09,8.999999E+09,8.999999E+09,8.999999E+09]];
    LOCAL CONST Robtarget Tr_meulage_motif_1_282 := [[-40.7026796875,180.710671875,32.584751953125],[0.205457264684473,-0.183019148705642,0.639481640238406,-0.717881978735665],[0,0,0,0],[8.999999E+09,8.999999E+09,8.999999E+09,8.999999E+09,8.999999E+09,8.999999E+09]];
    LOCAL CONST Robtarget Tr_meulage_motif_1_283 := [[-39.814515625,181.170203125,32.58475],[0.205457264684473,-0.183019148705642,0.639481640238406,-0.717881978735665],[0,0,0,0],[8.999999E+09,8.999999E+09,8.999999E+09,8.999999E+09,8.999999E+09,8.999999E+09]];
    LOCAL CONST Robtarget Tr_meulage_motif_1_284 := [[-38.9263515625,181.629734375,32.58475],[0.205457264684473,-0.183019148705642,0.639481640238406,-0.717881978735665],[0,0,0,0],[8.999999E+09,8.999999E+09,8.999999E+09,8.999999E+09,8.999999E+09,8.999999E+09]];
    LOCAL CONST Robtarget Tr_meulage_motif_1_285 := [[-38.0381875,182.08925,32.58475],[0.205457264684473,-0.183019148705642,0.639481640238406,-0.717881978735665],[0,0,0,0],[8.999999E+09,8.999999E+09,8.999999E+09,8.999999E+09,8.999999E+09,8.999999E+09]];
    LOCAL CONST Robtarget Tr_meulage_motif_1_286 := [[-37.1500234375,182.54878125,32.58475],[0.205457264684473,-0.183019148705642,0.639481640238406,-0.717881978735665],[0,0,0,0],[8.999999E+09,8.999999E+09,8.999999E+09,8.999999E+09,8.999999E+09,8.999999E+09]];
    LOCAL CONST Robtarget Tr_meulage_motif_1_287 := [[-36.261859375,183.0083125,32.58475],[0.205457264684473,-0.183019148705642,0.639481640238406,-0.717881978735665],[0,0,0,0],[8.999999E+09,8.999999E+09,8.999999E+09,8.999999E+09,8.999999E+09,8.999999E+09]];
    LOCAL CONST Robtarget Tr_meulage_motif_1_288 := [[-35.3736953125,183.46784375,32.584748046875],[0.205457264684473,-0.183019148705642,0.639481640238406,-0.717881978735665],[0,0,0,0],[8.999999E+09,8.999999E+09,8.999999E+09,8.999999E+09,8.999999E+09,8.999999E+09]];
    LOCAL CONST Robtarget Tr_meulage_motif_1_289 := [[-34.48553515625,183.927359375,32.584748046875],[0.205457264684473,-0.183019148705642,0.639481640238406,-0.717881978735665],[0,0,0,0],[8.999999E+09,8.999999E+09,8.999999E+09,8.999999E+09,8.999999E+09,8.999999E+09]];
    LOCAL CONST Robtarget Tr_meulage_motif_1_290 := [[-33.59737109375,184.386890625,32.584748046875],[0.205457264684473,-0.183019148705642,0.639481640238406,-0.717881978735665],[0,0,0,0],[8.999999E+09,8.999999E+09,8.999999E+09,8.999999E+09,8.999999E+09,8.999999E+09]];
    LOCAL CONST Robtarget Tr_meulage_motif_1_291 := [[-32.709205078125,184.846421875,32.584748046875],[0.205457264684473,-0.183019148705642,0.639481640238406,-0.717881978735665],[0,0,0,0],[8.999999E+09,8.999999E+09,8.999999E+09,8.999999E+09,8.999999E+09,8.999999E+09]];
    LOCAL CONST Robtarget Tr_meulage_motif_1_292 := [[-31.82104296875,185.305953125,32.58474609375],[0.205457264684473,-0.183019148705642,0.639481640238406,-0.717881978735665],[0,0,0,0],[8.999999E+09,8.999999E+09,8.999999E+09,8.999999E+09,8.999999E+09,8.999999E+09]];
    LOCAL CONST Robtarget Tr_meulage_motif_1_293 := [[-30.93287890625,185.76546875,32.58474609375],[0.205457264684473,-0.183019148705642,0.639481640238406,-0.717881978735665],[0,0,0,0],[8.999999E+09,8.999999E+09,8.999999E+09,8.999999E+09,8.999999E+09,8.999999E+09]];
    LOCAL CONST Robtarget Tr_meulage_motif_1_294 := [[-30.04471484375,186.225,32.58474609375],[0.205457264684473,-0.183019148705642,0.639481640238406,-0.717881978735665],[0,0,0,0],[8.999999E+09,8.999999E+09,8.999999E+09,8.999999E+09,8.999999E+09,8.999999E+09]];
    LOCAL CONST Robtarget Tr_meulage_motif_1_295 := [[-29.15655078125,186.68453125,32.58474609375],[0.205457264684473,-0.183019148705642,0.639481640238406,-0.717881978735665],[0,0,0,0],[8.999999E+09,8.999999E+09,8.999999E+09,8.999999E+09,8.999999E+09,8.999999E+09]];
    LOCAL CONST Robtarget Tr_meulage_motif_1_296 := [[-28.268388671875,187.1440625,32.584744140625],[0.205457264684473,-0.183019148705642,0.639481640238406,-0.717881978735665],[0,0,0,0],[8.999999E+09,8.999999E+09,8.999999E+09,8.999999E+09,8.999999E+09,8.999999E+09]];
    LOCAL CONST Robtarget Tr_meulage_motif_1_297 := [[-27.380224609375,187.603578125,32.584744140625],[0.205457264684473,-0.183019148705642,0.639481640238406,-0.717881978735665],[0,0,0,0],[8.999999E+09,8.999999E+09,8.999999E+09,8.999999E+09,8.999999E+09,8.999999E+09]];
    LOCAL CONST Robtarget Tr_meulage_motif_1_298 := [[-26.492060546875,188.063109375,32.584744140625],[0.205457264684473,-0.183019148705642,0.639481640238406,-0.717881978735665],[0,0,0,0],[8.999999E+09,8.999999E+09,8.999999E+09,8.999999E+09,8.999999E+09,8.999999E+09]];
    LOCAL CONST Robtarget Tr_meulage_motif_1_299 := [[-25.603896484375,188.522640625,32.584744140625],[0.205457264684473,-0.183019148705642,0.639481640238406,-0.717881978735665],[0,0,0,0],[8.999999E+09,8.999999E+09,8.999999E+09,8.999999E+09,8.999999E+09,8.999999E+09]];
    LOCAL CONST Robtarget Tr_meulage_motif_1_300 := [[-24.715734375,188.982171875,32.5847421875],[0.205457264684473,-0.183019148705642,0.639481640238406,-0.717881978735665],[0,0,0,0],[8.999999E+09,8.999999E+09,8.999999E+09,8.999999E+09,8.999999E+09,8.999999E+09]];
    LOCAL CONST Robtarget Tr_meulage_motif_1_301 := [[-23.8275703125,189.4416875,32.5847421875],[0.205457264684473,-0.183019148705642,0.639481640238406,-0.717881978735665],[0,0,0,0],[8.999999E+09,8.999999E+09,8.999999E+09,8.999999E+09,8.999999E+09,8.999999E+09]];
    LOCAL CONST Robtarget Tr_meulage_motif_1_302 := [[-22.93940625,189.90121875,32.5847421875],[0.205457264684473,-0.183019148705642,0.639481640238406,-0.717881978735665],[0,0,0,0],[8.999999E+09,8.999999E+09,8.999999E+09,8.999999E+09,8.999999E+09,8.999999E+09]];
    LOCAL CONST Robtarget Tr_meulage_motif_1_303 := [[-22.0512421875,190.36075,32.5847421875],[0.205457264684473,-0.183019148705642,0.639481640238406,-0.717881978735665],[0,0,0,0],[8.999999E+09,8.999999E+09,8.999999E+09,8.999999E+09,8.999999E+09,8.999999E+09]];
    LOCAL CONST Robtarget Tr_meulage_motif_1_304 := [[-21.163080078125,190.82028125,32.5847421875],[0.205457264684473,-0.183019148705642,0.639481640238406,-0.717881978735665],[0,0,0,0],[8.999999E+09,8.999999E+09,8.999999E+09,8.999999E+09,8.999999E+09,8.999999E+09]];
    LOCAL CONST Robtarget Tr_meulage_motif_1_305 := [[-20.274916015625,191.279796875,32.584740234375],[0.205457264684473,-0.183019148705642,0.639481640238406,-0.717881978735665],[0,0,0,0],[8.999999E+09,8.999999E+09,8.999999E+09,8.999999E+09,8.999999E+09,8.999999E+09]];
    LOCAL CONST Robtarget Tr_meulage_motif_1_306 := [[-19.386751953125,191.739328125,32.584740234375],[0.205457264684473,-0.183019148705642,0.639481640238406,-0.717881978735665],[0,0,0,0],[8.999999E+09,8.999999E+09,8.999999E+09,8.999999E+09,8.999999E+09,8.999999E+09]];
    LOCAL CONST Robtarget Tr_meulage_motif_1_307 := [[-18.498587890625,192.198859375,32.584740234375],[0.205457264684473,-0.183019148705642,0.639481640238406,-0.717881978735665],[0,0,0,0],[8.999999E+09,8.999999E+09,8.999999E+09,8.999999E+09,8.999999E+09,8.999999E+09]];
    LOCAL CONST Robtarget Tr_meulage_motif_1_308 := [[-17.61042578125,192.658390625,32.584740234375],[0.205457264684473,-0.183019148705642,0.639481640238406,-0.717881978735665],[0,0,0,0],[8.999999E+09,8.999999E+09,8.999999E+09,8.999999E+09,8.999999E+09,8.999999E+09]];
    LOCAL CONST Robtarget Tr_meulage_motif_1_309 := [[-16.72226171875,193.117921875,32.58473828125],[0.205457264684473,-0.183019148705642,0.639481640238406,-0.717881978735665],[0,0,0,0],[8.999999E+09,8.999999E+09,8.999999E+09,8.999999E+09,8.999999E+09,8.999999E+09]];
    LOCAL CONST Robtarget Tr_meulage_motif_1_310 := [[-15.83409765625,193.5774375,32.58473828125],[0.205457264684473,-0.183019148705642,0.639481640238406,-0.717881978735665],[0,0,0,0],[8.999999E+09,8.999999E+09,8.999999E+09,8.999999E+09,8.999999E+09,8.999999E+09]];
    LOCAL CONST Robtarget Tr_meulage_motif_1_311 := [[-14.9459345703125,194.03696875,32.58473828125],[0.205457264684473,-0.183019148705642,0.639481640238406,-0.717881978735665],[0,0,0,0],[8.999999E+09,8.999999E+09,8.999999E+09,8.999999E+09,8.999999E+09,8.999999E+09]];
    LOCAL CONST Robtarget Tr_meulage_motif_1_312 := [[-14.06478125,194.493859375,32.474146484375],[0.205457264684473,-0.183019148705642,0.639481640238406,-0.717881978735665],[0,0,0,0],[8.999999E+09,8.999999E+09,8.999999E+09,8.999999E+09,8.999999E+09,8.999999E+09]];
    LOCAL CONST Robtarget Tr_meulage_motif_1_313 := [[-13.2249072265625,194.930296875,32.262966796875],[0.205457264684473,-0.183019148705642,0.639481640238406,-0.717881978735665],[0,0,0,0],[8.999999E+09,8.999999E+09,8.999999E+09,8.999999E+09,8.999999E+09,8.999999E+09]];
    LOCAL CONST Robtarget Tr_meulage_motif_1_314 := [[-12.468548828125,195.3240625,31.991130859375],[0.205457264684473,-0.183019148705642,0.639481640238406,-0.717881978735665],[0,0,0,0],[8.999999E+09,8.999999E+09,8.999999E+09,8.999999E+09,8.999999E+09,8.999999E+09]];
    LOCAL CONST Robtarget Tr_meulage_motif_1_315 := [[-11.837734375,195.653171875,31.687],[0.205457264684473,-0.183019148705642,0.639481640238406,-0.717881978735665],[0,0,0,0],[8.999999E+09,8.999999E+09,8.999999E+09,8.999999E+09,8.999999E+09,8.999999E+09]];
    LOCAL CONST Robtarget Tr_meulage_motif_1_316 := [[-10.9213828125,196.133234375,31.02448828125],[0.205457264684473,-0.183019148705642,0.639481640238406,-0.717881978735665],[0,0,0,0],[8.999999E+09,8.999999E+09,8.999999E+09,8.999999E+09,8.999999E+09,8.999999E+09]];
    LOCAL CONST Robtarget Tr_meulage_motif_1_317 := [[-10.1236171875,196.554078125,30.122564453125],[0.205457264684473,-0.183019148705642,0.639481640238406,-0.717881978735665],[0,0,0,0],[8.999999E+09,8.999999E+09,8.999999E+09,8.999999E+09,8.999999E+09,8.999999E+09]];
    LOCAL CONST Robtarget Tr_meulage_motif_1_318 := [[-9.6523076171875,196.8073125,29.07658203125],[0.205457264684473,-0.183019148705642,0.639481640238406,-0.717881978735665],[0,0,0,0],[8.999999E+09,8.999999E+09,8.999999E+09,8.999999E+09,8.999999E+09,8.999999E+09]];
    LOCAL CONST Robtarget Tr_meulage_motif_1_319 := [[-9.49073046875,196.897125,28.383369140625],[0.205457264684473,-0.183019148705642,0.639481640238406,-0.717881978735665],[0,0,0,0],[8.999999E+09,8.999999E+09,8.999999E+09,8.999999E+09,8.999999E+09,8.999999E+09]];
    LOCAL CONST Robtarget Tr_meulage_motif_1_320 := [[-9.436845703125,196.931921875,27.613392578125],[0.205457264684473,-0.183019148705642,0.639481640238406,-0.717881978735665],[0,0,0,0],[8.999999E+09,8.999999E+09,8.999999E+09,8.999999E+09,8.999999E+09,8.999999E+09]];
    LOCAL CONST Robtarget Tr_meulage_motif_1_321 := [[-9.4991162109375,196.906609375,26.84355859375],[0.205457264684473,-0.183019148705642,0.639481640238406,-0.717881978735665],[0,0,0,0],[8.999999E+09,8.999999E+09,8.999999E+09,8.999999E+09,8.999999E+09,8.999999E+09]];
    LOCAL CONST Robtarget Tr_meulage_motif_1_322 := [[-9.875841796875,196.721625,25.73534375],[0.205457264684473,-0.183019148705642,0.639481640238406,-0.717881978735665],[0,0,0,0],[8.999999E+09,8.999999E+09,8.999999E+09,8.999999E+09,8.999999E+09,8.999999E+09]];
    LOCAL CONST Robtarget Tr_meulage_motif_1_323 := [[-10.2459638671875,196.535390625,25.149673828125],[0.205457264684473,-0.183019148705642,0.639481640238406,-0.717881978735665],[0,0,0,0],[8.999999E+09,8.999999E+09,8.999999E+09,8.999999E+09,8.999999E+09,8.999999E+09]];
    LOCAL CONST Robtarget Tr_meulage_motif_1_324 := [[-11.0371240234375,196.134,24.262546875],[0.205457264684473,-0.183019148705642,0.639481640238406,-0.717881978735665],[0,0,0,0],[8.999999E+09,8.999999E+09,8.999999E+09,8.999999E+09,8.999999E+09,8.999999E+09]];
    LOCAL CONST Robtarget Tr_meulage_motif_1_325 := [[-11.558828125,195.867796875,23.848279296875],[0.205457264684473,-0.183019148705642,0.639481640238406,-0.717881978735665],[0,0,0,0],[8.999999E+09,8.999999E+09,8.999999E+09,8.999999E+09,8.999999E+09,8.999999E+09]];
    LOCAL CONST Robtarget Tr_meulage_motif_1_326 := [[-12.5537041015625,195.3579375,23.304171875],[0.205457264684473,-0.183019148705642,0.639481640238406,-0.717881978735665],[0,0,0,0],[8.999999E+09,8.999999E+09,8.999999E+09,8.999999E+09,8.999999E+09,8.999999E+09]];
    LOCAL CONST Robtarget Tr_meulage_motif_1_327 := [[-13.2880478515625,194.980640625,23.008681640625],[0.205457264684473,-0.183019148705642,0.639481640238406,-0.717881978735665],[0,0,0,0],[8.999999E+09,8.999999E+09,8.999999E+09,8.999999E+09,8.999999E+09,8.999999E+09]];
    LOCAL CONST Robtarget Tr_meulage_motif_1_328 := [[-14.1165654296875,194.5538125,22.804205078125],[0.205457264684473,-0.183019148705642,0.639481640238406,-0.717881978735665],[0,0,0,0],[8.999999E+09,8.999999E+09,8.999999E+09,8.999999E+09,8.999999E+09,8.999999E+09]];
    LOCAL CONST Robtarget Tr_meulage_motif_1_329 := [[-14.9887509765625,194.10353125,22.695662109375],[0.205457264684473,-0.183019148705642,0.639481640238406,-0.717881978735665],[0,0,0,0],[8.999999E+09,8.999999E+09,8.999999E+09,8.999999E+09,8.999999E+09,8.999999E+09]];
    LOCAL CONST Robtarget Tr_meulage_motif_1_330 := [[-15.8707138671875,193.648203125,22.585056640625],[0.205457264684473,-0.183019148705642,0.639481640238406,-0.717881978735665],[0,0,0,0],[8.999999E+09,8.999999E+09,8.999999E+09,8.999999E+09,8.999999E+09,8.999999E+09]];
    LOCAL CONST Robtarget Tr_meulage_motif_1_331 := [[-16.758876953125,193.188671875,22.585056640625],[0.205457264684473,-0.183019148705642,0.639481640238406,-0.717881978735665],[0,0,0,0],[8.999999E+09,8.999999E+09,8.999999E+09,8.999999E+09,8.999999E+09,8.999999E+09]];
    LOCAL CONST Robtarget Tr_meulage_motif_1_332 := [[-17.647041015625,192.729140625,22.585056640625],[0.205457264684473,-0.183019148705642,0.639481640238406,-0.717881978735665],[0,0,0,0],[8.999999E+09,8.999999E+09,8.999999E+09,8.999999E+09,8.999999E+09,8.999999E+09]];
    LOCAL CONST Robtarget Tr_meulage_motif_1_333 := [[-18.535205078125,192.269625,22.585056640625],[0.205457264684473,-0.183019148705642,0.639481640238406,-0.717881978735665],[0,0,0,0],[8.999999E+09,8.999999E+09,8.999999E+09,8.999999E+09,8.999999E+09,8.999999E+09]];
    LOCAL CONST Robtarget Tr_meulage_motif_1_334 := [[-19.4233671875,191.81009375,22.58505859375],[0.205457264684473,-0.183019148705642,0.639481640238406,-0.717881978735665],[0,0,0,0],[8.999999E+09,8.999999E+09,8.999999E+09,8.999999E+09,8.999999E+09,8.999999E+09]];
    LOCAL CONST Robtarget Tr_meulage_motif_1_335 := [[-20.31153125,191.3505625,22.58505859375],[0.205457264684473,-0.183019148705642,0.639481640238406,-0.717881978735665],[0,0,0,0],[8.999999E+09,8.999999E+09,8.999999E+09,8.999999E+09,8.999999E+09,8.999999E+09]];
    LOCAL CONST Robtarget Tr_meulage_motif_1_336 := [[-21.1996953125,190.89103125,22.58505859375],[0.205457264684473,-0.183019148705642,0.639481640238406,-0.717881978735665],[0,0,0,0],[8.999999E+09,8.999999E+09,8.999999E+09,8.999999E+09,8.999999E+09,8.999999E+09]];
    LOCAL CONST Robtarget Tr_meulage_motif_1_337 := [[-22.087859375,190.431515625,22.58505859375],[0.205457264684473,-0.183019148705642,0.639481640238406,-0.717881978735665],[0,0,0,0],[8.999999E+09,8.999999E+09,8.999999E+09,8.999999E+09,8.999999E+09,8.999999E+09]];
    LOCAL CONST Robtarget Tr_meulage_motif_1_338 := [[-22.976021484375,189.971984375,22.585060546875],[0.205457264684473,-0.183019148705642,0.639481640238406,-0.717881978735665],[0,0,0,0],[8.999999E+09,8.999999E+09,8.999999E+09,8.999999E+09,8.999999E+09,8.999999E+09]];
    LOCAL CONST Robtarget Tr_meulage_motif_1_339 := [[-23.864185546875,189.512453125,22.585060546875],[0.205457264684473,-0.183019148705642,0.639481640238406,-0.717881978735665],[0,0,0,0],[8.999999E+09,8.999999E+09,8.999999E+09,8.999999E+09,8.999999E+09,8.999999E+09]];
    LOCAL CONST Robtarget Tr_meulage_motif_1_340 := [[-24.752349609375,189.052921875,22.585060546875],[0.205457264684473,-0.183019148705642,0.639481640238406,-0.717881978735665],[0,0,0,0],[8.999999E+09,8.999999E+09,8.999999E+09,8.999999E+09,8.999999E+09,8.999999E+09]];
    LOCAL CONST Robtarget Tr_meulage_motif_1_341 := [[-25.640513671875,188.59340625,22.585060546875],[0.205457264684473,-0.183019148705642,0.639481640238406,-0.717881978735665],[0,0,0,0],[8.999999E+09,8.999999E+09,8.999999E+09,8.999999E+09,8.999999E+09,8.999999E+09]];
    LOCAL CONST Robtarget Tr_meulage_motif_1_342 := [[-26.52867578125,188.133875,22.585060546875],[0.205457264684473,-0.183019148705642,0.639481640238406,-0.717881978735665],[0,0,0,0],[8.999999E+09,8.999999E+09,8.999999E+09,8.999999E+09,8.999999E+09,8.999999E+09]];
    LOCAL CONST Robtarget Tr_meulage_motif_1_343 := [[-27.41683984375,187.67434375,22.5850625],[0.205457264684473,-0.183019148705642,0.639481640238406,-0.717881978735665],[0,0,0,0],[8.999999E+09,8.999999E+09,8.999999E+09,8.999999E+09,8.999999E+09,8.999999E+09]];
    LOCAL CONST Robtarget Tr_meulage_motif_1_344 := [[-28.30500390625,187.2148125,22.5850625],[0.205457264684473,-0.183019148705642,0.639481640238406,-0.717881978735665],[0,0,0,0],[8.999999E+09,8.999999E+09,8.999999E+09,8.999999E+09,8.999999E+09,8.999999E+09]];
    LOCAL CONST Robtarget Tr_meulage_motif_1_345 := [[-29.19316796875,186.755296875,22.5850625],[0.205457264684473,-0.183019148705642,0.639481640238406,-0.717881978735665],[0,0,0,0],[8.999999E+09,8.999999E+09,8.999999E+09,8.999999E+09,8.999999E+09,8.999999E+09]];
    LOCAL CONST Robtarget Tr_meulage_motif_1_346 := [[-30.08133203125,186.295765625,22.5850625],[0.205457264684473,-0.183019148705642,0.639481640238406,-0.717881978735665],[0,0,0,0],[8.999999E+09,8.999999E+09,8.999999E+09,8.999999E+09,8.999999E+09,8.999999E+09]];
    LOCAL CONST Robtarget Tr_meulage_motif_1_347 := [[-30.969494140625,185.836234375,22.585064453125],[0.205457264684473,-0.183019148705642,0.639481640238406,-0.717881978735665],[0,0,0,0],[8.999999E+09,8.999999E+09,8.999999E+09,8.999999E+09,8.999999E+09,8.999999E+09]];
    LOCAL CONST Robtarget Tr_meulage_motif_1_348 := [[-31.857658203125,185.376703125,22.585064453125],[0.205457264684473,-0.183019148705642,0.639481640238406,-0.717881978735665],[0,0,0,0],[8.999999E+09,8.999999E+09,8.999999E+09,8.999999E+09,8.999999E+09,8.999999E+09]];
    LOCAL CONST Robtarget Tr_meulage_motif_1_349 := [[-32.745822265625,184.9171875,22.585064453125],[0.205457264684473,-0.183019148705642,0.639481640238406,-0.717881978735665],[0,0,0,0],[8.999999E+09,8.999999E+09,8.999999E+09,8.999999E+09,8.999999E+09,8.999999E+09]];
    LOCAL CONST Robtarget Tr_meulage_motif_1_350 := [[-33.633984375,184.45765625,22.585064453125],[0.205457264684473,-0.183019148705642,0.639481640238406,-0.717881978735665],[0,0,0,0],[8.999999E+09,8.999999E+09,8.999999E+09,8.999999E+09,8.999999E+09,8.999999E+09]];
    LOCAL CONST Robtarget Tr_meulage_motif_1_351 := [[-34.5221484375,183.998125,22.58506640625],[0.205457264684473,-0.183019148705642,0.639481640238406,-0.717881978735665],[0,0,0,0],[8.999999E+09,8.999999E+09,8.999999E+09,8.999999E+09,8.999999E+09,8.999999E+09]];
    LOCAL CONST Robtarget Tr_meulage_motif_1_352 := [[-35.4103125,183.53859375,22.58506640625],[0.205457264684473,-0.183019148705642,0.639481640238406,-0.717881978735665],[0,0,0,0],[8.999999E+09,8.999999E+09,8.999999E+09,8.999999E+09,8.999999E+09,8.999999E+09]];
    LOCAL CONST Robtarget Tr_meulage_motif_1_353 := [[-36.2984765625,183.079078125,22.58506640625],[0.205457264684473,-0.183019148705642,0.639481640238406,-0.717881978735665],[0,0,0,0],[8.999999E+09,8.999999E+09,8.999999E+09,8.999999E+09,8.999999E+09,8.999999E+09]];
    LOCAL CONST Robtarget Tr_meulage_motif_1_354 := [[-37.186640625,182.619546875,22.58506640625],[0.205457264684473,-0.183019148705642,0.639481640238406,-0.717881978735665],[0,0,0,0],[8.999999E+09,8.999999E+09,8.999999E+09,8.999999E+09,8.999999E+09,8.999999E+09]];
    LOCAL CONST Robtarget Tr_meulage_motif_1_355 := [[-38.0748046875,182.160015625,22.58506640625],[0.205457264684473,-0.183019148705642,0.639481640238406,-0.717881978735665],[0,0,0,0],[8.999999E+09,8.999999E+09,8.999999E+09,8.999999E+09,8.999999E+09,8.999999E+09]];
    LOCAL CONST Robtarget Tr_meulage_motif_1_356 := [[-38.96296875,181.700484375,22.585068359375],[0.205457264684473,-0.183019148705642,0.639481640238406,-0.717881978735665],[0,0,0,0],[8.999999E+09,8.999999E+09,8.999999E+09,8.999999E+09,8.999999E+09,8.999999E+09]];
    LOCAL CONST Robtarget Tr_meulage_motif_1_357 := [[-39.85112890625,181.24096875,22.585068359375],[0.205457264684473,-0.183019148705642,0.639481640238406,-0.717881978735665],[0,0,0,0],[8.999999E+09,8.999999E+09,8.999999E+09,8.999999E+09,8.999999E+09,8.999999E+09]];
    LOCAL CONST Robtarget Tr_meulage_motif_1_358 := [[-40.73929296875,180.7814375,22.585068359375],[0.205457264684473,-0.183019148705642,0.639481640238406,-0.717881978735665],[0,0,0,0],[8.999999E+09,8.999999E+09,8.999999E+09,8.999999E+09,8.999999E+09,8.999999E+09]];
    LOCAL CONST Robtarget Tr_meulage_motif_1_359 := [[-41.62745703125,180.32190625,22.585068359375],[0.205457264684473,-0.183019148705642,0.639481640238406,-0.717881978735665],[0,0,0,0],[8.999999E+09,8.999999E+09,8.999999E+09,8.999999E+09,8.999999E+09,8.999999E+09]];
    LOCAL CONST Robtarget Tr_meulage_motif_1_360 := [[-42.51562109375,179.862375,22.5850703125],[0.205457264684473,-0.183019148705642,0.639481640238406,-0.717881978735665],[0,0,0,0],[8.999999E+09,8.999999E+09,8.999999E+09,8.999999E+09,8.999999E+09,8.999999E+09]];
    LOCAL CONST Robtarget Tr_meulage_motif_1_361 := [[-43.40378515625,179.402859375,22.5850703125],[0.205457264684473,-0.183019148705642,0.639481640238406,-0.717881978735665],[0,0,0,0],[8.999999E+09,8.999999E+09,8.999999E+09,8.999999E+09,8.999999E+09,8.999999E+09]];
    LOCAL CONST Robtarget Tr_meulage_motif_1_362 := [[-44.29194921875,178.943328125,22.5850703125],[0.205457264684473,-0.183019148705642,0.639481640238406,-0.717881978735665],[0,0,0,0],[8.999999E+09,8.999999E+09,8.999999E+09,8.999999E+09,8.999999E+09,8.999999E+09]];
    LOCAL CONST Robtarget Tr_meulage_motif_1_363 := [[-45.18011328125,178.483796875,22.5850703125],[0.205457264684473,-0.183019148705642,0.639481640238406,-0.717881978735665],[0,0,0,0],[8.999999E+09,8.999999E+09,8.999999E+09,8.999999E+09,8.999999E+09,8.999999E+09]];
    LOCAL CONST Robtarget Tr_meulage_motif_1_364 := [[-46.06827734375,178.024265625,22.585072265625],[0.205457264684473,-0.183019148705642,0.639481640238406,-0.717881978735665],[0,0,0,0],[8.999999E+09,8.999999E+09,8.999999E+09,8.999999E+09,8.999999E+09,8.999999E+09]];
    LOCAL CONST Robtarget Tr_meulage_motif_1_365 := [[-46.95644140625,177.56475,22.585072265625],[0.205457264684473,-0.183019148705642,0.639481640238406,-0.717881978735665],[0,0,0,0],[8.999999E+09,8.999999E+09,8.999999E+09,8.999999E+09,8.999999E+09,8.999999E+09]];
    LOCAL CONST Robtarget Tr_meulage_motif_1_366 := [[-47.8446015625,177.10521875,22.585072265625],[0.205457264684473,-0.183019148705642,0.639481640238406,-0.717881978735665],[0,0,0,0],[8.999999E+09,8.999999E+09,8.999999E+09,8.999999E+09,8.999999E+09,8.999999E+09]];
    LOCAL CONST Robtarget Tr_meulage_motif_1_367 := [[-48.732765625,176.6456875,22.585072265625],[0.205457264684473,-0.183019148705642,0.639481640238406,-0.717881978735665],[0,0,0,0],[8.999999E+09,8.999999E+09,8.999999E+09,8.999999E+09,8.999999E+09,8.999999E+09]];
    LOCAL CONST Robtarget Tr_meulage_motif_1_368 := [[-49.6209296875,176.18615625,22.58507421875],[0.205457264684473,-0.183019148705642,0.639481640238406,-0.717881978735665],[0,0,0,0],[8.999999E+09,8.999999E+09,8.999999E+09,8.999999E+09,8.999999E+09,8.999999E+09]];
    LOCAL CONST Robtarget Tr_meulage_motif_1_369 := [[-50.50909375,175.726640625,22.58507421875],[0.205457264684473,-0.183019148705642,0.639481640238406,-0.717881978735665],[0,0,0,0],[8.999999E+09,8.999999E+09,8.999999E+09,8.999999E+09,8.999999E+09,8.999999E+09]];
    LOCAL CONST Robtarget Tr_meulage_motif_1_370 := [[-51.3972578125,175.267109375,22.58507421875],[0.205457264684473,-0.183019148705642,0.639481640238406,-0.717881978735665],[0,0,0,0],[8.999999E+09,8.999999E+09,8.999999E+09,8.999999E+09,8.999999E+09,8.999999E+09]];
    LOCAL CONST Robtarget Tr_meulage_motif_1_371 := [[-52.285421875,174.807578125,22.58507421875],[0.205457264684473,-0.183019148705642,0.639481640238406,-0.717881978735665],[0,0,0,0],[8.999999E+09,8.999999E+09,8.999999E+09,8.999999E+09,8.999999E+09,8.999999E+09]];
